// TIA Portal V18 export
// export: Created 2025-12-01T17:51:00.4461215Z, ExportSetting None, DisplayName Totally Integrated Automation Portal, DisplayVersion V18 Update 5, DisplayName TIA Portal Openness, DisplayVersion V18 Update 5, DisplayName TIA Portal Teamcenter Gateway, DisplayVersion V18, DisplayName TIA Portal Version Control Interface, DisplayVersion V18, DisplayName STEP 7 Professional, DisplayVersion V18 Update 5, DisplayName STEP 7 Safety, DisplayVersion V18, DisplayName WinCC Professional, DisplayVersion V18 Update 5
DATA_BLOCK "Parameter"   // DB170
{ S7_Optimized_Access := 'TRUE' }
// stored: AutoNumber false, IsRetainMemResEnabled true, MemoryReserve 10000
   VAR RETAIN
      AxisRun : Struct
         Axis : Array[1..15] of "ServoType_UDT";
      END_STRUCT;
      AxisNuw : Struct
         Axis : Array[1..15] of "ServoType_UDT";
      END_STRUCT;
      AxisDisplay : Struct
         Axis : Array[1..15] of "ServoType_UDT";
      END_STRUCT;
      AxisSave : Struct
         Axis : Array[1..15] of "ServoType_UDT";
      END_STRUCT;
      AxisStore : Array[1..15] of Struct
         Axis : Array[1..15] of "ServoType_UDT";
      END_STRUCT;
   END_VAR
BEGIN
   // AxisRun.Axis[1].Pos1 : 上料位1
   // AxisRun.Axis[2].Pos1 : 初始位
   // AxisRun.Axis[3].Pos1 : Home position / IV camera position 1
   // AxisRun.Axis[4].Pos1 : 上料位1
   // AxisRun.Axis[5].Pos1 : Z轴初始位
   // AxisRun.Axis[6].Pos1 : X轴初始位
   // AxisRun.Axis[7].Pos1 : Y轴初始位
   AxisRun.Axis[1].Pos1.Position := 3.12;
   AxisRun.Axis[2..3].Pos1.Position := 0.0;
   AxisRun.Axis[4].Pos1.Position := 3.585;
   AxisRun.Axis[5].Pos1.Position := 143.76;
   AxisRun.Axis[6].Pos1.Position := 2.34;
   AxisRun.Axis[7].Pos1.Position := 115.47;
   AxisRun.Axis[8..15].Pos1.Position := 0.0;
   AxisRun.Axis[1..2].Pos1.Speed := 10000;
   AxisRun.Axis[3].Pos1.Speed := 20000;
   AxisRun.Axis[4].Pos1.Speed := 10000;
   AxisRun.Axis[5..7].Pos1.Speed := 200;
   AxisRun.Axis[8..15].Pos1.Speed := 0;
   AxisRun.Axis[1..15].Pos1.Reached := FALSE;
   // AxisRun.Axis[1].Pos2 : 上料位2
   // AxisRun.Axis[2].Pos2 : 扫码位置2
   // AxisRun.Axis[3].Pos2 : Glue station 1 – end position
   // AxisRun.Axis[4].Pos2 : 上料位2
   // AxisRun.Axis[5].Pos2 : Z轴点胶位1
   // AxisRun.Axis[6].Pos2 : X轴点胶等待位
   // AxisRun.Axis[7].Pos2 : Y轴点胶位1
   AxisRun.Axis[1].Pos2.Position := 48.058;
   AxisRun.Axis[2].Pos2.Position := 45.0;
   AxisRun.Axis[3].Pos2.Position := 490.0;
   AxisRun.Axis[4].Pos2.Position := 48.61;
   AxisRun.Axis[5].Pos2.Position := 139.11;
   AxisRun.Axis[6].Pos2.Position := 76.0;
   AxisRun.Axis[7].Pos2.Position := 115.47;
   AxisRun.Axis[8..15].Pos2.Position := 0.0;
   AxisRun.Axis[1..2].Pos2.Speed := 10000;
   AxisRun.Axis[3].Pos2.Speed := 20000;
   AxisRun.Axis[4].Pos2.Speed := 10000;
   AxisRun.Axis[5..7].Pos2.Speed := 200;
   AxisRun.Axis[8..15].Pos2.Speed := 0;
   AxisRun.Axis[1..15].Pos2.Reached := FALSE;
   // AxisRun.Axis[1].Pos3 : 上料位3
   // AxisRun.Axis[2].Pos3 : 扫码位置3
   // AxisRun.Axis[3].Pos3 : Glue station 2 – end position
   // AxisRun.Axis[4].Pos3 : 上料位3
   // AxisRun.Axis[5].Pos3 : Z轴点胶位2
   // AxisRun.Axis[6].Pos3 : X轴点胶位1
   // AxisRun.Axis[7].Pos3 : Y轴点胶位2
   AxisRun.Axis[1].Pos3.Position := 93.154;
   AxisRun.Axis[2].Pos3.Position := 90.0;
   AxisRun.Axis[3].Pos3.Position := 490.0;
   AxisRun.Axis[4].Pos3.Position := 93.637;
   AxisRun.Axis[5].Pos3.Position := 131.98;
   AxisRun.Axis[6].Pos3.Position := 84.69;
   AxisRun.Axis[7].Pos3.Position := 115.47;
   AxisRun.Axis[8..15].Pos3.Position := 0.0;
   AxisRun.Axis[1..2].Pos3.Speed := 10000;
   AxisRun.Axis[3].Pos3.Speed := 20000;
   AxisRun.Axis[4].Pos3.Speed := 10000;
   AxisRun.Axis[5..7].Pos3.Speed := 200;
   AxisRun.Axis[8..15].Pos3.Speed := 0;
   AxisRun.Axis[1..15].Pos3.Reached := FALSE;
   // AxisRun.Axis[1].Pos4 : 上料位4
   // AxisRun.Axis[2].Pos4 : 扫码位置4
   // AxisRun.Axis[3].Pos4 : Glue station 3 – end position
   // AxisRun.Axis[4].Pos4 : 上料位4
   // AxisRun.Axis[5].Pos4 : Z轴点胶位3
   // AxisRun.Axis[6].Pos4 : X轴点胶位2
   // AxisRun.Axis[7].Pos4 : Y轴点胶位3
   AxisRun.Axis[1].Pos4.Position := 138.111;
   AxisRun.Axis[2].Pos4.Position := 135.0;
   AxisRun.Axis[3].Pos4.Position := 490.0;
   AxisRun.Axis[4].Pos4.Position := 138.606;
   AxisRun.Axis[5].Pos4.Position := 127.89;
   AxisRun.Axis[6].Pos4.Position := 84.69;
   AxisRun.Axis[7].Pos4.Position := 115.47;
   AxisRun.Axis[8..15].Pos4.Position := 0.0;
   AxisRun.Axis[1..2].Pos4.Speed := 10000;
   AxisRun.Axis[3].Pos4.Speed := 20000;
   AxisRun.Axis[4].Pos4.Speed := 10000;
   AxisRun.Axis[5..7].Pos4.Speed := 200;
   AxisRun.Axis[8..15].Pos4.Speed := 0;
   AxisRun.Axis[1..15].Pos4.Reached := FALSE;
   // AxisRun.Axis[1].Pos5 : 上料位5
   // AxisRun.Axis[2].Pos5 : 扫码位置5
   // AxisRun.Axis[3].Pos5 : Glue station 4 – end position // glue position cancelled
   // AxisRun.Axis[4].Pos5 : 上料位5
   // AxisRun.Axis[5].Pos5 : Z轴点胶位4
   // AxisRun.Axis[6].Pos5 : X轴点胶位3
   // AxisRun.Axis[7].Pos5 : Y轴点胶位4
   AxisRun.Axis[1].Pos5.Position := 183.025;
   AxisRun.Axis[2].Pos5.Position := 180.0;
   AxisRun.Axis[3].Pos5.Position := 0.0;
   AxisRun.Axis[4].Pos5.Position := 183.388;
   AxisRun.Axis[5].Pos5.Position := 0.0;
   AxisRun.Axis[6].Pos5.Position := 84.69;
   AxisRun.Axis[7].Pos5.Position := 115.47;
   AxisRun.Axis[8..15].Pos5.Position := 0.0;
   AxisRun.Axis[1..2].Pos5.Speed := 10000;
   AxisRun.Axis[3].Pos5.Speed := 0;
   AxisRun.Axis[4].Pos5.Speed := 10000;
   AxisRun.Axis[5].Pos5.Speed := 0;
   AxisRun.Axis[6..7].Pos5.Speed := 200;
   AxisRun.Axis[8..15].Pos5.Speed := 0;
   AxisRun.Axis[1..15].Pos5.Reached := FALSE;
   // AxisRun.Axis[1].Pos6 : 上料位6
   // AxisRun.Axis[2].Pos6 : 扫码位置6
   // AxisRun.Axis[3].Pos6 : Glue station 5 – end position
   // AxisRun.Axis[4].Pos6 : 上料位6
   // AxisRun.Axis[5].Pos6 : Z轴点胶位5
   // AxisRun.Axis[6].Pos6 : X轴点胶位4
   // AxisRun.Axis[7].Pos6 : Y轴点胶位5
   AxisRun.Axis[1].Pos6.Position := 228.065;
   AxisRun.Axis[2].Pos6.Position := 225.0;
   AxisRun.Axis[3].Pos6.Position := 490.0;
   AxisRun.Axis[4].Pos6.Position := 228.458;
   AxisRun.Axis[5].Pos6.Position := 127.0;
   AxisRun.Axis[6].Pos6.Position := 84.69;
   AxisRun.Axis[7].Pos6.Position := 110.18;
   AxisRun.Axis[8..15].Pos6.Position := 0.0;
   AxisRun.Axis[1..2].Pos6.Speed := 10000;
   AxisRun.Axis[3].Pos6.Speed := 5000;
   AxisRun.Axis[4].Pos6.Speed := 10000;
   AxisRun.Axis[5..7].Pos6.Speed := 200;
   AxisRun.Axis[8..15].Pos6.Speed := 0;
   AxisRun.Axis[1..15].Pos6.Reached := FALSE;
   // AxisRun.Axis[1].Pos7 : 上料位7
   // AxisRun.Axis[2].Pos7 : 扫码位置7
   // AxisRun.Axis[3].Pos7 : IV camera position 2
   // AxisRun.Axis[4].Pos7 : 上料位7
   // AxisRun.Axis[5].Pos7 : Z轴相机检测位
   // AxisRun.Axis[6].Pos7 : X轴点胶位5
   // AxisRun.Axis[7].Pos7 : Y轴相机检测位
   AxisRun.Axis[1].Pos7.Position := 273.195;
   AxisRun.Axis[2].Pos7.Position := 270.0;
   AxisRun.Axis[3].Pos7.Position := 90.0;
   AxisRun.Axis[4].Pos7.Position := 273.513;
   AxisRun.Axis[5].Pos7.Position := 48.11;
   AxisRun.Axis[6].Pos7.Position := 85.0;
   AxisRun.Axis[7].Pos7.Position := 60.52;
   AxisRun.Axis[8..15].Pos7.Position := 0.0;
   AxisRun.Axis[1..2].Pos7.Speed := 10000;
   AxisRun.Axis[3].Pos7.Speed := 20000;
   AxisRun.Axis[4].Pos7.Speed := 10000;
   AxisRun.Axis[5..7].Pos7.Speed := 200;
   AxisRun.Axis[8..15].Pos7.Speed := 0;
   AxisRun.Axis[1..15].Pos7.Reached := FALSE;
   // AxisRun.Axis[1].Pos8 : 上料位8
   // AxisRun.Axis[2].Pos8 : 扫码位置8
   // AxisRun.Axis[3].Pos8 : IV camera position 3
   // AxisRun.Axis[4].Pos8 : 上料位8
   // AxisRun.Axis[5].Pos8 : Z轴原点位
   // AxisRun.Axis[6].Pos8 : X轴相机检测位
   AxisRun.Axis[1].Pos8.Position := 318.05;
   AxisRun.Axis[2].Pos8.Position := 315.0;
   AxisRun.Axis[3].Pos8.Position := 180.0;
   AxisRun.Axis[4].Pos8.Position := 318.501;
   AxisRun.Axis[5].Pos8.Position := 0.0;
   AxisRun.Axis[6].Pos8.Position := 88.53;
   AxisRun.Axis[7].Pos8.Position := 80.0;
   AxisRun.Axis[8..15].Pos8.Position := 0.0;
   AxisRun.Axis[1..2].Pos8.Speed := 10000;
   AxisRun.Axis[3].Pos8.Speed := 20000;
   AxisRun.Axis[4].Pos8.Speed := 10000;
   AxisRun.Axis[5..6].Pos8.Speed := 200;
   AxisRun.Axis[7].Pos8.Speed := 100;
   AxisRun.Axis[8..15].Pos8.Speed := 0;
   AxisRun.Axis[1..15].Pos8.Reached := FALSE;
   // AxisRun.Axis[3].Pos9 : IV camera position 4
   // AxisRun.Axis[5].Pos9 : Z轴Up点胶位5
   AxisRun.Axis[1..2].Pos9.Position := 0.0;
   AxisRun.Axis[3].Pos9.Position := 270.0;
   AxisRun.Axis[4].Pos9.Position := 0.0;
   AxisRun.Axis[5].Pos9.Position := 48.11;
   AxisRun.Axis[6..15].Pos9.Position := 0.0;
   AxisRun.Axis[1..2].Pos9.Speed := 0;
   AxisRun.Axis[3].Pos9.Speed := 20000;
   AxisRun.Axis[4].Pos9.Speed := 0;
   AxisRun.Axis[5].Pos9.Speed := 200;
   AxisRun.Axis[6..15].Pos9.Speed := 0;
   AxisRun.Axis[1..15].Pos9.Reached := FALSE;
   AxisRun.Axis[1..15].Pos10.Position := 0.0;
   AxisRun.Axis[1..15].Pos10.Speed := 0;
   AxisRun.Axis[1..15].Pos10.Reached := FALSE;
   AxisRun.Axis[1..15].Pos11.Position := 0.0;
   AxisRun.Axis[1..15].Pos11.Speed := 0;
   AxisRun.Axis[1..15].Pos11.Reached := FALSE;
   AxisRun.Axis[1..15].Pos12.Position := 0.0;
   AxisRun.Axis[1..15].Pos12.Speed := 0;
   AxisRun.Axis[1..15].Pos12.Reached := FALSE;
   AxisRun.Axis[1..15].Pos13.Position := 0.0;
   AxisRun.Axis[1..15].Pos13.Speed := 0;
   AxisRun.Axis[1..15].Pos13.Reached := FALSE;
   AxisRun.Axis[1..15].Pos14.Position := 0.0;
   AxisRun.Axis[1..15].Pos14.Speed := 0;
   AxisRun.Axis[1..15].Pos14.Reached := FALSE;
   AxisRun.Axis[1..15].Pos15.Position := 0.0;
   AxisRun.Axis[1..15].Pos15.Speed := 0;
   AxisRun.Axis[1..15].Pos15.Reached := FALSE;
   AxisRun.Axis[1..15].Pos16.Position := 0.0;
   AxisRun.Axis[1..15].Pos16.Speed := 0;
   AxisRun.Axis[1..15].Pos16.Reached := FALSE;
   AxisRun.Axis[1..15].Pos17.Position := 0.0;
   AxisRun.Axis[1..15].Pos17.Speed := 0;
   AxisRun.Axis[1..15].Pos17.Reached := FALSE;
   AxisRun.Axis[1..15].Pos18.Position := 0.0;
   AxisRun.Axis[1..15].Pos18.Speed := 0;
   AxisRun.Axis[1..15].Pos18.Reached := FALSE;
   AxisRun.Axis[1..15].Pos19.Position := 0.0;
   AxisRun.Axis[1..15].Pos19.Speed := 0;
   AxisRun.Axis[1..15].Pos19.Reached := FALSE;
   AxisRun.Axis[1..15].Pos20.Position := 0.0;
   AxisRun.Axis[1..15].Pos20.Speed := 0;
   AxisRun.Axis[1..15].Pos20.Reached := FALSE;
   AxisRun.Axis[1..15].Pos21.Position := 0.0;
   AxisRun.Axis[1..15].Pos21.Speed := 0;
   AxisRun.Axis[1..15].Pos21.Reached := FALSE;
   AxisRun.Axis[1..15].Pos22.Position := 0.0;
   AxisRun.Axis[1..15].Pos22.Speed := 0;
   AxisRun.Axis[1..15].Pos22.Reached := FALSE;
   AxisRun.Axis[1..15].Pos23.Position := 0.0;
   AxisRun.Axis[1..15].Pos23.Speed := 0;
   AxisRun.Axis[1..15].Pos23.Reached := FALSE;
   AxisRun.Axis[1..15].Pos24.Position := 0.0;
   AxisRun.Axis[1..15].Pos24.Speed := 0;
   AxisRun.Axis[1..15].Pos24.Reached := FALSE;
   AxisRun.Axis[1..15].Pos25.Position := 0.0;
   AxisRun.Axis[1..15].Pos25.Speed := 0;
   AxisRun.Axis[1..15].Pos25.Reached := FALSE;
   AxisRun.Axis[1..15].Pos26.Position := 0.0;
   AxisRun.Axis[1..15].Pos26.Speed := 0;
   AxisRun.Axis[1..15].Pos26.Reached := FALSE;
   AxisRun.Axis[1..15].Pos27.Position := 0.0;
   AxisRun.Axis[1..15].Pos27.Speed := 0;
   AxisRun.Axis[1..15].Pos27.Reached := FALSE;
   AxisRun.Axis[1..15].Pos28.Position := 0.0;
   AxisRun.Axis[1..15].Pos28.Speed := 0;
   AxisRun.Axis[1..15].Pos28.Reached := FALSE;
   AxisRun.Axis[1..15].Pos29.Position := 0.0;
   AxisRun.Axis[1..15].Pos29.Speed := 0;
   AxisRun.Axis[1..15].Pos29.Reached := FALSE;
   AxisRun.Axis[1..15].Pos30.Position := 0.0;
   AxisRun.Axis[1..15].Pos30.Speed := 0;
   AxisRun.Axis[1..15].Pos30.Reached := FALSE;
   AxisNuw.Axis[1..15].Pos1.Position := 0.0;
   AxisNuw.Axis[1..15].Pos1.Speed := 0;
   AxisNuw.Axis[1..15].Pos1.Reached := FALSE;
   AxisNuw.Axis[1..15].Pos2.Position := 0.0;
   AxisNuw.Axis[1..15].Pos2.Speed := 0;
   AxisNuw.Axis[1..15].Pos2.Reached := FALSE;
   AxisNuw.Axis[1..15].Pos3.Position := 0.0;
   AxisNuw.Axis[1..15].Pos3.Speed := 0;
   AxisNuw.Axis[1..15].Pos3.Reached := FALSE;
   AxisNuw.Axis[1..15].Pos4.Position := 0.0;
   AxisNuw.Axis[1..15].Pos4.Speed := 0;
   AxisNuw.Axis[1..15].Pos4.Reached := FALSE;
   AxisNuw.Axis[1..15].Pos5.Position := 0.0;
   AxisNuw.Axis[1..15].Pos5.Speed := 0;
   AxisNuw.Axis[1..15].Pos5.Reached := FALSE;
   AxisNuw.Axis[1..15].Pos6.Position := 0.0;
   AxisNuw.Axis[1..15].Pos6.Speed := 0;
   AxisNuw.Axis[1..15].Pos6.Reached := FALSE;
   AxisNuw.Axis[1..15].Pos7.Position := 0.0;
   AxisNuw.Axis[1..15].Pos7.Speed := 0;
   AxisNuw.Axis[1..15].Pos7.Reached := FALSE;
   AxisNuw.Axis[1..15].Pos8.Position := 0.0;
   AxisNuw.Axis[1..15].Pos8.Speed := 0;
   AxisNuw.Axis[1..15].Pos8.Reached := FALSE;
   AxisNuw.Axis[1..15].Pos9.Position := 0.0;
   AxisNuw.Axis[1..15].Pos9.Speed := 0;
   AxisNuw.Axis[1..15].Pos9.Reached := FALSE;
   AxisNuw.Axis[1..15].Pos10.Position := 0.0;
   AxisNuw.Axis[1..15].Pos10.Speed := 0;
   AxisNuw.Axis[1..15].Pos10.Reached := FALSE;
   AxisNuw.Axis[1..15].Pos11.Position := 0.0;
   AxisNuw.Axis[1..15].Pos11.Speed := 0;
   AxisNuw.Axis[1..15].Pos11.Reached := FALSE;
   AxisNuw.Axis[1..15].Pos12.Position := 0.0;
   AxisNuw.Axis[1..15].Pos12.Speed := 0;
   AxisNuw.Axis[1..15].Pos12.Reached := FALSE;
   AxisNuw.Axis[1..15].Pos13.Position := 0.0;
   AxisNuw.Axis[1..15].Pos13.Speed := 0;
   AxisNuw.Axis[1..15].Pos13.Reached := FALSE;
   AxisNuw.Axis[1..15].Pos14.Position := 0.0;
   AxisNuw.Axis[1..15].Pos14.Speed := 0;
   AxisNuw.Axis[1..15].Pos14.Reached := FALSE;
   AxisNuw.Axis[1..15].Pos15.Position := 0.0;
   AxisNuw.Axis[1..15].Pos15.Speed := 0;
   AxisNuw.Axis[1..15].Pos15.Reached := FALSE;
   AxisNuw.Axis[1..15].Pos16.Position := 0.0;
   AxisNuw.Axis[1..15].Pos16.Speed := 0;
   AxisNuw.Axis[1..15].Pos16.Reached := FALSE;
   AxisNuw.Axis[1..15].Pos17.Position := 0.0;
   AxisNuw.Axis[1..15].Pos17.Speed := 0;
   AxisNuw.Axis[1..15].Pos17.Reached := FALSE;
   AxisNuw.Axis[1..15].Pos18.Position := 0.0;
   AxisNuw.Axis[1..15].Pos18.Speed := 0;
   AxisNuw.Axis[1..15].Pos18.Reached := FALSE;
   AxisNuw.Axis[1..15].Pos19.Position := 0.0;
   AxisNuw.Axis[1..15].Pos19.Speed := 0;
   AxisNuw.Axis[1..15].Pos19.Reached := FALSE;
   AxisNuw.Axis[1..15].Pos20.Position := 0.0;
   AxisNuw.Axis[1..15].Pos20.Speed := 0;
   AxisNuw.Axis[1..15].Pos20.Reached := FALSE;
   AxisNuw.Axis[1..15].Pos21.Position := 0.0;
   AxisNuw.Axis[1..15].Pos21.Speed := 0;
   AxisNuw.Axis[1..15].Pos21.Reached := FALSE;
   AxisNuw.Axis[1..15].Pos22.Position := 0.0;
   AxisNuw.Axis[1..15].Pos22.Speed := 0;
   AxisNuw.Axis[1..15].Pos22.Reached := FALSE;
   AxisNuw.Axis[1..15].Pos23.Position := 0.0;
   AxisNuw.Axis[1..15].Pos23.Speed := 0;
   AxisNuw.Axis[1..15].Pos23.Reached := FALSE;
   AxisNuw.Axis[1..15].Pos24.Position := 0.0;
   AxisNuw.Axis[1..15].Pos24.Speed := 0;
   AxisNuw.Axis[1..15].Pos24.Reached := FALSE;
   AxisNuw.Axis[1..15].Pos25.Position := 0.0;
   AxisNuw.Axis[1..15].Pos25.Speed := 0;
   AxisNuw.Axis[1..15].Pos25.Reached := FALSE;
   AxisNuw.Axis[1..15].Pos26.Position := 0.0;
   AxisNuw.Axis[1..15].Pos26.Speed := 0;
   AxisNuw.Axis[1..15].Pos26.Reached := FALSE;
   AxisNuw.Axis[1..15].Pos27.Position := 0.0;
   AxisNuw.Axis[1..15].Pos27.Speed := 0;
   AxisNuw.Axis[1..15].Pos27.Reached := FALSE;
   AxisNuw.Axis[1..15].Pos28.Position := 0.0;
   AxisNuw.Axis[1..15].Pos28.Speed := 0;
   AxisNuw.Axis[1..15].Pos28.Reached := FALSE;
   AxisNuw.Axis[1..15].Pos29.Position := 0.0;
   AxisNuw.Axis[1..15].Pos29.Speed := 0;
   AxisNuw.Axis[1..15].Pos29.Reached := FALSE;
   AxisNuw.Axis[1..15].Pos30.Position := 0.0;
   AxisNuw.Axis[1..15].Pos30.Speed := 0;
   AxisNuw.Axis[1..15].Pos30.Reached := FALSE;
   AxisDisplay.Axis[1..15].Pos1.Position := 0.0;
   AxisDisplay.Axis[1..15].Pos1.Speed := 0;
   AxisDisplay.Axis[1..15].Pos1.Reached := FALSE;
   AxisDisplay.Axis[1..15].Pos2.Position := 0.0;
   AxisDisplay.Axis[1..15].Pos2.Speed := 0;
   AxisDisplay.Axis[1..15].Pos2.Reached := FALSE;
   AxisDisplay.Axis[1..15].Pos3.Position := 0.0;
   AxisDisplay.Axis[1..15].Pos3.Speed := 0;
   AxisDisplay.Axis[1..15].Pos3.Reached := FALSE;
   AxisDisplay.Axis[1..15].Pos4.Position := 0.0;
   AxisDisplay.Axis[1..15].Pos4.Speed := 0;
   AxisDisplay.Axis[1..15].Pos4.Reached := FALSE;
   AxisDisplay.Axis[1..15].Pos5.Position := 0.0;
   AxisDisplay.Axis[1..15].Pos5.Speed := 0;
   AxisDisplay.Axis[1..15].Pos5.Reached := FALSE;
   AxisDisplay.Axis[1..15].Pos6.Position := 0.0;
   AxisDisplay.Axis[1..15].Pos6.Speed := 0;
   AxisDisplay.Axis[1..15].Pos6.Reached := FALSE;
   AxisDisplay.Axis[1..15].Pos7.Position := 0.0;
   AxisDisplay.Axis[1..15].Pos7.Speed := 0;
   AxisDisplay.Axis[1..15].Pos7.Reached := FALSE;
   AxisDisplay.Axis[1..15].Pos8.Position := 0.0;
   AxisDisplay.Axis[1..15].Pos8.Speed := 0;
   AxisDisplay.Axis[1..15].Pos8.Reached := FALSE;
   AxisDisplay.Axis[1..15].Pos9.Position := 0.0;
   AxisDisplay.Axis[1..15].Pos9.Speed := 0;
   AxisDisplay.Axis[1..15].Pos9.Reached := FALSE;
   AxisDisplay.Axis[1..15].Pos10.Position := 0.0;
   AxisDisplay.Axis[1..15].Pos10.Speed := 0;
   AxisDisplay.Axis[1..15].Pos10.Reached := FALSE;
   AxisDisplay.Axis[1..15].Pos11.Position := 0.0;
   AxisDisplay.Axis[1..15].Pos11.Speed := 0;
   AxisDisplay.Axis[1..15].Pos11.Reached := FALSE;
   AxisDisplay.Axis[1..15].Pos12.Position := 0.0;
   AxisDisplay.Axis[1..15].Pos12.Speed := 0;
   AxisDisplay.Axis[1..15].Pos12.Reached := FALSE;
   AxisDisplay.Axis[1..15].Pos13.Position := 0.0;
   AxisDisplay.Axis[1..15].Pos13.Speed := 0;
   AxisDisplay.Axis[1..15].Pos13.Reached := FALSE;
   AxisDisplay.Axis[1..15].Pos14.Position := 0.0;
   AxisDisplay.Axis[1..15].Pos14.Speed := 0;
   AxisDisplay.Axis[1..15].Pos14.Reached := FALSE;
   AxisDisplay.Axis[1..15].Pos15.Position := 0.0;
   AxisDisplay.Axis[1..15].Pos15.Speed := 0;
   AxisDisplay.Axis[1..15].Pos15.Reached := FALSE;
   AxisDisplay.Axis[1..15].Pos16.Position := 0.0;
   AxisDisplay.Axis[1..15].Pos16.Speed := 0;
   AxisDisplay.Axis[1..15].Pos16.Reached := FALSE;
   AxisDisplay.Axis[1..15].Pos17.Position := 0.0;
   AxisDisplay.Axis[1..15].Pos17.Speed := 0;
   AxisDisplay.Axis[1..15].Pos17.Reached := FALSE;
   AxisDisplay.Axis[1..15].Pos18.Position := 0.0;
   AxisDisplay.Axis[1..15].Pos18.Speed := 0;
   AxisDisplay.Axis[1..15].Pos18.Reached := FALSE;
   AxisDisplay.Axis[1..15].Pos19.Position := 0.0;
   AxisDisplay.Axis[1..15].Pos19.Speed := 0;
   AxisDisplay.Axis[1..15].Pos19.Reached := FALSE;
   AxisDisplay.Axis[1..15].Pos20.Position := 0.0;
   AxisDisplay.Axis[1..15].Pos20.Speed := 0;
   AxisDisplay.Axis[1..15].Pos20.Reached := FALSE;
   AxisDisplay.Axis[1..15].Pos21.Position := 0.0;
   AxisDisplay.Axis[1..15].Pos21.Speed := 0;
   AxisDisplay.Axis[1..15].Pos21.Reached := FALSE;
   AxisDisplay.Axis[1..15].Pos22.Position := 0.0;
   AxisDisplay.Axis[1..15].Pos22.Speed := 0;
   AxisDisplay.Axis[1..15].Pos22.Reached := FALSE;
   AxisDisplay.Axis[1..15].Pos23.Position := 0.0;
   AxisDisplay.Axis[1..15].Pos23.Speed := 0;
   AxisDisplay.Axis[1..15].Pos23.Reached := FALSE;
   AxisDisplay.Axis[1..15].Pos24.Position := 0.0;
   AxisDisplay.Axis[1..15].Pos24.Speed := 0;
   AxisDisplay.Axis[1..15].Pos24.Reached := FALSE;
   AxisDisplay.Axis[1..15].Pos25.Position := 0.0;
   AxisDisplay.Axis[1..15].Pos25.Speed := 0;
   AxisDisplay.Axis[1..15].Pos25.Reached := FALSE;
   AxisDisplay.Axis[1..15].Pos26.Position := 0.0;
   AxisDisplay.Axis[1..15].Pos26.Speed := 0;
   AxisDisplay.Axis[1..15].Pos26.Reached := FALSE;
   AxisDisplay.Axis[1..15].Pos27.Position := 0.0;
   AxisDisplay.Axis[1..15].Pos27.Speed := 0;
   AxisDisplay.Axis[1..15].Pos27.Reached := FALSE;
   AxisDisplay.Axis[1..15].Pos28.Position := 0.0;
   AxisDisplay.Axis[1..15].Pos28.Speed := 0;
   AxisDisplay.Axis[1..15].Pos28.Reached := FALSE;
   AxisDisplay.Axis[1..15].Pos29.Position := 0.0;
   AxisDisplay.Axis[1..15].Pos29.Speed := 0;
   AxisDisplay.Axis[1..15].Pos29.Reached := FALSE;
   AxisDisplay.Axis[1..15].Pos30.Position := 0.0;
   AxisDisplay.Axis[1..15].Pos30.Speed := 0;
   AxisDisplay.Axis[1..15].Pos30.Reached := FALSE;
   AxisSave.Axis[1..15].Pos1.Position := 0.0;
   AxisSave.Axis[1..15].Pos1.Speed := 0;
   AxisSave.Axis[1..15].Pos1.Reached := FALSE;
   AxisSave.Axis[1..15].Pos2.Position := 0.0;
   AxisSave.Axis[1..15].Pos2.Speed := 0;
   AxisSave.Axis[1..15].Pos2.Reached := FALSE;
   AxisSave.Axis[1..15].Pos3.Position := 0.0;
   AxisSave.Axis[1..15].Pos3.Speed := 0;
   AxisSave.Axis[1..15].Pos3.Reached := FALSE;
   AxisSave.Axis[1..15].Pos4.Position := 0.0;
   AxisSave.Axis[1..15].Pos4.Speed := 0;
   AxisSave.Axis[1..15].Pos4.Reached := FALSE;
   AxisSave.Axis[1..15].Pos5.Position := 0.0;
   AxisSave.Axis[1..15].Pos5.Speed := 0;
   AxisSave.Axis[1..15].Pos5.Reached := FALSE;
   AxisSave.Axis[1..15].Pos6.Position := 0.0;
   AxisSave.Axis[1..15].Pos6.Speed := 0;
   AxisSave.Axis[1..15].Pos6.Reached := FALSE;
   AxisSave.Axis[1..15].Pos7.Position := 0.0;
   AxisSave.Axis[1..15].Pos7.Speed := 0;
   AxisSave.Axis[1..15].Pos7.Reached := FALSE;
   AxisSave.Axis[1..15].Pos8.Position := 0.0;
   AxisSave.Axis[1..15].Pos8.Speed := 0;
   AxisSave.Axis[1..15].Pos8.Reached := FALSE;
   AxisSave.Axis[1..15].Pos9.Position := 0.0;
   AxisSave.Axis[1..15].Pos9.Speed := 0;
   AxisSave.Axis[1..15].Pos9.Reached := FALSE;
   AxisSave.Axis[1..15].Pos10.Position := 0.0;
   AxisSave.Axis[1..15].Pos10.Speed := 0;
   AxisSave.Axis[1..15].Pos10.Reached := FALSE;
   AxisSave.Axis[1..15].Pos11.Position := 0.0;
   AxisSave.Axis[1..15].Pos11.Speed := 0;
   AxisSave.Axis[1..15].Pos11.Reached := FALSE;
   AxisSave.Axis[1..15].Pos12.Position := 0.0;
   AxisSave.Axis[1..15].Pos12.Speed := 0;
   AxisSave.Axis[1..15].Pos12.Reached := FALSE;
   AxisSave.Axis[1..15].Pos13.Position := 0.0;
   AxisSave.Axis[1..15].Pos13.Speed := 0;
   AxisSave.Axis[1..15].Pos13.Reached := FALSE;
   AxisSave.Axis[1..15].Pos14.Position := 0.0;
   AxisSave.Axis[1..15].Pos14.Speed := 0;
   AxisSave.Axis[1..15].Pos14.Reached := FALSE;
   AxisSave.Axis[1..15].Pos15.Position := 0.0;
   AxisSave.Axis[1..15].Pos15.Speed := 0;
   AxisSave.Axis[1..15].Pos15.Reached := FALSE;
   AxisSave.Axis[1..15].Pos16.Position := 0.0;
   AxisSave.Axis[1..15].Pos16.Speed := 0;
   AxisSave.Axis[1..15].Pos16.Reached := FALSE;
   AxisSave.Axis[1..15].Pos17.Position := 0.0;
   AxisSave.Axis[1..15].Pos17.Speed := 0;
   AxisSave.Axis[1..15].Pos17.Reached := FALSE;
   AxisSave.Axis[1..15].Pos18.Position := 0.0;
   AxisSave.Axis[1..15].Pos18.Speed := 0;
   AxisSave.Axis[1..15].Pos18.Reached := FALSE;
   AxisSave.Axis[1..15].Pos19.Position := 0.0;
   AxisSave.Axis[1..15].Pos19.Speed := 0;
   AxisSave.Axis[1..15].Pos19.Reached := FALSE;
   AxisSave.Axis[1..15].Pos20.Position := 0.0;
   AxisSave.Axis[1..15].Pos20.Speed := 0;
   AxisSave.Axis[1..15].Pos20.Reached := FALSE;
   AxisSave.Axis[1..15].Pos21.Position := 0.0;
   AxisSave.Axis[1..15].Pos21.Speed := 0;
   AxisSave.Axis[1..15].Pos21.Reached := FALSE;
   AxisSave.Axis[1..15].Pos22.Position := 0.0;
   AxisSave.Axis[1..15].Pos22.Speed := 0;
   AxisSave.Axis[1..15].Pos22.Reached := FALSE;
   AxisSave.Axis[1..15].Pos23.Position := 0.0;
   AxisSave.Axis[1..15].Pos23.Speed := 0;
   AxisSave.Axis[1..15].Pos23.Reached := FALSE;
   AxisSave.Axis[1..15].Pos24.Position := 0.0;
   AxisSave.Axis[1..15].Pos24.Speed := 0;
   AxisSave.Axis[1..15].Pos24.Reached := FALSE;
   AxisSave.Axis[1..15].Pos25.Position := 0.0;
   AxisSave.Axis[1..15].Pos25.Speed := 0;
   AxisSave.Axis[1..15].Pos25.Reached := FALSE;
   AxisSave.Axis[1..15].Pos26.Position := 0.0;
   AxisSave.Axis[1..15].Pos26.Speed := 0;
   AxisSave.Axis[1..15].Pos26.Reached := FALSE;
   AxisSave.Axis[1..15].Pos27.Position := 0.0;
   AxisSave.Axis[1..15].Pos27.Speed := 0;
   AxisSave.Axis[1..15].Pos27.Reached := FALSE;
   AxisSave.Axis[1..15].Pos28.Position := 0.0;
   AxisSave.Axis[1..15].Pos28.Speed := 0;
   AxisSave.Axis[1..15].Pos28.Reached := FALSE;
   AxisSave.Axis[1..15].Pos29.Position := 0.0;
   AxisSave.Axis[1..15].Pos29.Speed := 0;
   AxisSave.Axis[1..15].Pos29.Reached := FALSE;
   AxisSave.Axis[1..15].Pos30.Position := 0.0;
   AxisSave.Axis[1..15].Pos30.Speed := 0;
   AxisSave.Axis[1..15].Pos30.Reached := FALSE;
   AxisStore[1].Axis[1..15].Pos1.Position := 0.0;
   AxisStore[2].Axis[1..15].Pos1.Position := 0.0;
   AxisStore[3].Axis[1..15].Pos1.Position := 0.0;
   AxisStore[4].Axis[1..15].Pos1.Position := 0.0;
   AxisStore[5].Axis[1..15].Pos1.Position := 0.0;
   AxisStore[6].Axis[1..15].Pos1.Position := 0.0;
   AxisStore[7].Axis[1..15].Pos1.Position := 0.0;
   AxisStore[8].Axis[1..15].Pos1.Position := 0.0;
   AxisStore[9].Axis[1..15].Pos1.Position := 0.0;
   AxisStore[10].Axis[1..15].Pos1.Position := 0.0;
   AxisStore[11].Axis[1..15].Pos1.Position := 0.0;
   AxisStore[12].Axis[1..15].Pos1.Position := 0.0;
   AxisStore[13].Axis[1..15].Pos1.Position := 0.0;
   AxisStore[14].Axis[1..15].Pos1.Position := 0.0;
   AxisStore[15].Axis[1..15].Pos1.Position := 0.0;
   AxisStore[1].Axis[1..15].Pos1.Speed := 0;
   AxisStore[2].Axis[1..15].Pos1.Speed := 0;
   AxisStore[3].Axis[1..15].Pos1.Speed := 0;
   AxisStore[4].Axis[1..15].Pos1.Speed := 0;
   AxisStore[5].Axis[1..15].Pos1.Speed := 0;
   AxisStore[6].Axis[1..15].Pos1.Speed := 0;
   AxisStore[7].Axis[1..15].Pos1.Speed := 0;
   AxisStore[8].Axis[1..15].Pos1.Speed := 0;
   AxisStore[9].Axis[1..15].Pos1.Speed := 0;
   AxisStore[10].Axis[1..15].Pos1.Speed := 0;
   AxisStore[11].Axis[1..15].Pos1.Speed := 0;
   AxisStore[12].Axis[1..15].Pos1.Speed := 0;
   AxisStore[13].Axis[1..15].Pos1.Speed := 0;
   AxisStore[14].Axis[1..15].Pos1.Speed := 0;
   AxisStore[15].Axis[1..15].Pos1.Speed := 0;
   AxisStore[1].Axis[1..15].Pos1.Reached := FALSE;
   AxisStore[2].Axis[1..15].Pos1.Reached := FALSE;
   AxisStore[3].Axis[1..15].Pos1.Reached := FALSE;
   AxisStore[4].Axis[1..15].Pos1.Reached := FALSE;
   AxisStore[5].Axis[1..15].Pos1.Reached := FALSE;
   AxisStore[6].Axis[1..15].Pos1.Reached := FALSE;
   AxisStore[7].Axis[1..15].Pos1.Reached := FALSE;
   AxisStore[8].Axis[1..15].Pos1.Reached := FALSE;
   AxisStore[9].Axis[1..15].Pos1.Reached := FALSE;
   AxisStore[10].Axis[1..15].Pos1.Reached := FALSE;
   AxisStore[11].Axis[1..15].Pos1.Reached := FALSE;
   AxisStore[12].Axis[1..15].Pos1.Reached := FALSE;
   AxisStore[13].Axis[1..15].Pos1.Reached := FALSE;
   AxisStore[14].Axis[1..15].Pos1.Reached := FALSE;
   AxisStore[15].Axis[1..15].Pos1.Reached := FALSE;
   AxisStore[1].Axis[1..15].Pos2.Position := 0.0;
   AxisStore[2].Axis[1..15].Pos2.Position := 0.0;
   AxisStore[3].Axis[1..15].Pos2.Position := 0.0;
   AxisStore[4].Axis[1..15].Pos2.Position := 0.0;
   AxisStore[5].Axis[1..15].Pos2.Position := 0.0;
   AxisStore[6].Axis[1..15].Pos2.Position := 0.0;
   AxisStore[7].Axis[1..15].Pos2.Position := 0.0;
   AxisStore[8].Axis[1..15].Pos2.Position := 0.0;
   AxisStore[9].Axis[1..15].Pos2.Position := 0.0;
   AxisStore[10].Axis[1..15].Pos2.Position := 0.0;
   AxisStore[11].Axis[1..15].Pos2.Position := 0.0;
   AxisStore[12].Axis[1..15].Pos2.Position := 0.0;
   AxisStore[13].Axis[1..15].Pos2.Position := 0.0;
   AxisStore[14].Axis[1..15].Pos2.Position := 0.0;
   AxisStore[15].Axis[1..15].Pos2.Position := 0.0;
   AxisStore[1].Axis[1..15].Pos2.Speed := 0;
   AxisStore[2].Axis[1..15].Pos2.Speed := 0;
   AxisStore[3].Axis[1..15].Pos2.Speed := 0;
   AxisStore[4].Axis[1..15].Pos2.Speed := 0;
   AxisStore[5].Axis[1..15].Pos2.Speed := 0;
   AxisStore[6].Axis[1..15].Pos2.Speed := 0;
   AxisStore[7].Axis[1..15].Pos2.Speed := 0;
   AxisStore[8].Axis[1..15].Pos2.Speed := 0;
   AxisStore[9].Axis[1..15].Pos2.Speed := 0;
   AxisStore[10].Axis[1..15].Pos2.Speed := 0;
   AxisStore[11].Axis[1..15].Pos2.Speed := 0;
   AxisStore[12].Axis[1..15].Pos2.Speed := 0;
   AxisStore[13].Axis[1..15].Pos2.Speed := 0;
   AxisStore[14].Axis[1..15].Pos2.Speed := 0;
   AxisStore[15].Axis[1..15].Pos2.Speed := 0;
   AxisStore[1].Axis[1..15].Pos2.Reached := FALSE;
   AxisStore[2].Axis[1..15].Pos2.Reached := FALSE;
   AxisStore[3].Axis[1..15].Pos2.Reached := FALSE;
   AxisStore[4].Axis[1..15].Pos2.Reached := FALSE;
   AxisStore[5].Axis[1..15].Pos2.Reached := FALSE;
   AxisStore[6].Axis[1..15].Pos2.Reached := FALSE;
   AxisStore[7].Axis[1..15].Pos2.Reached := FALSE;
   AxisStore[8].Axis[1..15].Pos2.Reached := FALSE;
   AxisStore[9].Axis[1..15].Pos2.Reached := FALSE;
   AxisStore[10].Axis[1..15].Pos2.Reached := FALSE;
   AxisStore[11].Axis[1..15].Pos2.Reached := FALSE;
   AxisStore[12].Axis[1..15].Pos2.Reached := FALSE;
   AxisStore[13].Axis[1..15].Pos2.Reached := FALSE;
   AxisStore[14].Axis[1..15].Pos2.Reached := FALSE;
   AxisStore[15].Axis[1..15].Pos2.Reached := FALSE;
   AxisStore[1].Axis[1..15].Pos3.Position := 0.0;
   AxisStore[2].Axis[1..15].Pos3.Position := 0.0;
   AxisStore[3].Axis[1..15].Pos3.Position := 0.0;
   AxisStore[4].Axis[1..15].Pos3.Position := 0.0;
   AxisStore[5].Axis[1..15].Pos3.Position := 0.0;
   AxisStore[6].Axis[1..15].Pos3.Position := 0.0;
   AxisStore[7].Axis[1..15].Pos3.Position := 0.0;
   AxisStore[8].Axis[1..15].Pos3.Position := 0.0;
   AxisStore[9].Axis[1..15].Pos3.Position := 0.0;
   AxisStore[10].Axis[1..15].Pos3.Position := 0.0;
   AxisStore[11].Axis[1..15].Pos3.Position := 0.0;
   AxisStore[12].Axis[1..15].Pos3.Position := 0.0;
   AxisStore[13].Axis[1..15].Pos3.Position := 0.0;
   AxisStore[14].Axis[1..15].Pos3.Position := 0.0;
   AxisStore[15].Axis[1..15].Pos3.Position := 0.0;
   AxisStore[1].Axis[1..15].Pos3.Speed := 0;
   AxisStore[2].Axis[1..15].Pos3.Speed := 0;
   AxisStore[3].Axis[1..15].Pos3.Speed := 0;
   AxisStore[4].Axis[1..15].Pos3.Speed := 0;
   AxisStore[5].Axis[1..15].Pos3.Speed := 0;
   AxisStore[6].Axis[1..15].Pos3.Speed := 0;
   AxisStore[7].Axis[1..15].Pos3.Speed := 0;
   AxisStore[8].Axis[1..15].Pos3.Speed := 0;
   AxisStore[9].Axis[1..15].Pos3.Speed := 0;
   AxisStore[10].Axis[1..15].Pos3.Speed := 0;
   AxisStore[11].Axis[1..15].Pos3.Speed := 0;
   AxisStore[12].Axis[1..15].Pos3.Speed := 0;
   AxisStore[13].Axis[1..15].Pos3.Speed := 0;
   AxisStore[14].Axis[1..15].Pos3.Speed := 0;
   AxisStore[15].Axis[1..15].Pos3.Speed := 0;
   AxisStore[1].Axis[1..15].Pos3.Reached := FALSE;
   AxisStore[2].Axis[1..15].Pos3.Reached := FALSE;
   AxisStore[3].Axis[1..15].Pos3.Reached := FALSE;
   AxisStore[4].Axis[1..15].Pos3.Reached := FALSE;
   AxisStore[5].Axis[1..15].Pos3.Reached := FALSE;
   AxisStore[6].Axis[1..15].Pos3.Reached := FALSE;
   AxisStore[7].Axis[1..15].Pos3.Reached := FALSE;
   AxisStore[8].Axis[1..15].Pos3.Reached := FALSE;
   AxisStore[9].Axis[1..15].Pos3.Reached := FALSE;
   AxisStore[10].Axis[1..15].Pos3.Reached := FALSE;
   AxisStore[11].Axis[1..15].Pos3.Reached := FALSE;
   AxisStore[12].Axis[1..15].Pos3.Reached := FALSE;
   AxisStore[13].Axis[1..15].Pos3.Reached := FALSE;
   AxisStore[14].Axis[1..15].Pos3.Reached := FALSE;
   AxisStore[15].Axis[1..15].Pos3.Reached := FALSE;
   AxisStore[1].Axis[1..15].Pos4.Position := 0.0;
   AxisStore[2].Axis[1..15].Pos4.Position := 0.0;
   AxisStore[3].Axis[1..15].Pos4.Position := 0.0;
   AxisStore[4].Axis[1..15].Pos4.Position := 0.0;
   AxisStore[5].Axis[1..15].Pos4.Position := 0.0;
   AxisStore[6].Axis[1..15].Pos4.Position := 0.0;
   AxisStore[7].Axis[1..15].Pos4.Position := 0.0;
   AxisStore[8].Axis[1..15].Pos4.Position := 0.0;
   AxisStore[9].Axis[1..15].Pos4.Position := 0.0;
   AxisStore[10].Axis[1..15].Pos4.Position := 0.0;
   AxisStore[11].Axis[1..15].Pos4.Position := 0.0;
   AxisStore[12].Axis[1..15].Pos4.Position := 0.0;
   AxisStore[13].Axis[1..15].Pos4.Position := 0.0;
   AxisStore[14].Axis[1..15].Pos4.Position := 0.0;
   AxisStore[15].Axis[1..15].Pos4.Position := 0.0;
   AxisStore[1].Axis[1..15].Pos4.Speed := 0;
   AxisStore[2].Axis[1..15].Pos4.Speed := 0;
   AxisStore[3].Axis[1..15].Pos4.Speed := 0;
   AxisStore[4].Axis[1..15].Pos4.Speed := 0;
   AxisStore[5].Axis[1..15].Pos4.Speed := 0;
   AxisStore[6].Axis[1..15].Pos4.Speed := 0;
   AxisStore[7].Axis[1..15].Pos4.Speed := 0;
   AxisStore[8].Axis[1..15].Pos4.Speed := 0;
   AxisStore[9].Axis[1..15].Pos4.Speed := 0;
   AxisStore[10].Axis[1..15].Pos4.Speed := 0;
   AxisStore[11].Axis[1..15].Pos4.Speed := 0;
   AxisStore[12].Axis[1..15].Pos4.Speed := 0;
   AxisStore[13].Axis[1..15].Pos4.Speed := 0;
   AxisStore[14].Axis[1..15].Pos4.Speed := 0;
   AxisStore[15].Axis[1..15].Pos4.Speed := 0;
   AxisStore[1].Axis[1..15].Pos4.Reached := FALSE;
   AxisStore[2].Axis[1..15].Pos4.Reached := FALSE;
   AxisStore[3].Axis[1..15].Pos4.Reached := FALSE;
   AxisStore[4].Axis[1..15].Pos4.Reached := FALSE;
   AxisStore[5].Axis[1..15].Pos4.Reached := FALSE;
   AxisStore[6].Axis[1..15].Pos4.Reached := FALSE;
   AxisStore[7].Axis[1..15].Pos4.Reached := FALSE;
   AxisStore[8].Axis[1..15].Pos4.Reached := FALSE;
   AxisStore[9].Axis[1..15].Pos4.Reached := FALSE;
   AxisStore[10].Axis[1..15].Pos4.Reached := FALSE;
   AxisStore[11].Axis[1..15].Pos4.Reached := FALSE;
   AxisStore[12].Axis[1..15].Pos4.Reached := FALSE;
   AxisStore[13].Axis[1..15].Pos4.Reached := FALSE;
   AxisStore[14].Axis[1..15].Pos4.Reached := FALSE;
   AxisStore[15].Axis[1..15].Pos4.Reached := FALSE;
   AxisStore[1].Axis[1..15].Pos5.Position := 0.0;
   AxisStore[2].Axis[1..15].Pos5.Position := 0.0;
   AxisStore[3].Axis[1..15].Pos5.Position := 0.0;
   AxisStore[4].Axis[1..15].Pos5.Position := 0.0;
   AxisStore[5].Axis[1..15].Pos5.Position := 0.0;
   AxisStore[6].Axis[1..15].Pos5.Position := 0.0;
   AxisStore[7].Axis[1..15].Pos5.Position := 0.0;
   AxisStore[8].Axis[1..15].Pos5.Position := 0.0;
   AxisStore[9].Axis[1..15].Pos5.Position := 0.0;
   AxisStore[10].Axis[1..15].Pos5.Position := 0.0;
   AxisStore[11].Axis[1..15].Pos5.Position := 0.0;
   AxisStore[12].Axis[1..15].Pos5.Position := 0.0;
   AxisStore[13].Axis[1..15].Pos5.Position := 0.0;
   AxisStore[14].Axis[1..15].Pos5.Position := 0.0;
   AxisStore[15].Axis[1..15].Pos5.Position := 0.0;
   AxisStore[1].Axis[1..15].Pos5.Speed := 0;
   AxisStore[2].Axis[1..15].Pos5.Speed := 0;
   AxisStore[3].Axis[1..15].Pos5.Speed := 0;
   AxisStore[4].Axis[1..15].Pos5.Speed := 0;
   AxisStore[5].Axis[1..15].Pos5.Speed := 0;
   AxisStore[6].Axis[1..15].Pos5.Speed := 0;
   AxisStore[7].Axis[1..15].Pos5.Speed := 0;
   AxisStore[8].Axis[1..15].Pos5.Speed := 0;
   AxisStore[9].Axis[1..15].Pos5.Speed := 0;
   AxisStore[10].Axis[1..15].Pos5.Speed := 0;
   AxisStore[11].Axis[1..15].Pos5.Speed := 0;
   AxisStore[12].Axis[1..15].Pos5.Speed := 0;
   AxisStore[13].Axis[1..15].Pos5.Speed := 0;
   AxisStore[14].Axis[1..15].Pos5.Speed := 0;
   AxisStore[15].Axis[1..15].Pos5.Speed := 0;
   AxisStore[1].Axis[1..15].Pos5.Reached := FALSE;
   AxisStore[2].Axis[1..15].Pos5.Reached := FALSE;
   AxisStore[3].Axis[1..15].Pos5.Reached := FALSE;
   AxisStore[4].Axis[1..15].Pos5.Reached := FALSE;
   AxisStore[5].Axis[1..15].Pos5.Reached := FALSE;
   AxisStore[6].Axis[1..15].Pos5.Reached := FALSE;
   AxisStore[7].Axis[1..15].Pos5.Reached := FALSE;
   AxisStore[8].Axis[1..15].Pos5.Reached := FALSE;
   AxisStore[9].Axis[1..15].Pos5.Reached := FALSE;
   AxisStore[10].Axis[1..15].Pos5.Reached := FALSE;
   AxisStore[11].Axis[1..15].Pos5.Reached := FALSE;
   AxisStore[12].Axis[1..15].Pos5.Reached := FALSE;
   AxisStore[13].Axis[1..15].Pos5.Reached := FALSE;
   AxisStore[14].Axis[1..15].Pos5.Reached := FALSE;
   AxisStore[15].Axis[1..15].Pos5.Reached := FALSE;
   AxisStore[1].Axis[1..15].Pos6.Position := 0.0;
   AxisStore[2].Axis[1..15].Pos6.Position := 0.0;
   AxisStore[3].Axis[1..15].Pos6.Position := 0.0;
   AxisStore[4].Axis[1..15].Pos6.Position := 0.0;
   AxisStore[5].Axis[1..15].Pos6.Position := 0.0;
   AxisStore[6].Axis[1..15].Pos6.Position := 0.0;
   AxisStore[7].Axis[1..15].Pos6.Position := 0.0;
   AxisStore[8].Axis[1..15].Pos6.Position := 0.0;
   AxisStore[9].Axis[1..15].Pos6.Position := 0.0;
   AxisStore[10].Axis[1..15].Pos6.Position := 0.0;
   AxisStore[11].Axis[1..15].Pos6.Position := 0.0;
   AxisStore[12].Axis[1..15].Pos6.Position := 0.0;
   AxisStore[13].Axis[1..15].Pos6.Position := 0.0;
   AxisStore[14].Axis[1..15].Pos6.Position := 0.0;
   AxisStore[15].Axis[1..15].Pos6.Position := 0.0;
   AxisStore[1].Axis[1..15].Pos6.Speed := 0;
   AxisStore[2].Axis[1..15].Pos6.Speed := 0;
   AxisStore[3].Axis[1..15].Pos6.Speed := 0;
   AxisStore[4].Axis[1..15].Pos6.Speed := 0;
   AxisStore[5].Axis[1..15].Pos6.Speed := 0;
   AxisStore[6].Axis[1..15].Pos6.Speed := 0;
   AxisStore[7].Axis[1..15].Pos6.Speed := 0;
   AxisStore[8].Axis[1..15].Pos6.Speed := 0;
   AxisStore[9].Axis[1..15].Pos6.Speed := 0;
   AxisStore[10].Axis[1..15].Pos6.Speed := 0;
   AxisStore[11].Axis[1..15].Pos6.Speed := 0;
   AxisStore[12].Axis[1..15].Pos6.Speed := 0;
   AxisStore[13].Axis[1..15].Pos6.Speed := 0;
   AxisStore[14].Axis[1..15].Pos6.Speed := 0;
   AxisStore[15].Axis[1..15].Pos6.Speed := 0;
   AxisStore[1].Axis[1..15].Pos6.Reached := FALSE;
   AxisStore[2].Axis[1..15].Pos6.Reached := FALSE;
   AxisStore[3].Axis[1..15].Pos6.Reached := FALSE;
   AxisStore[4].Axis[1..15].Pos6.Reached := FALSE;
   AxisStore[5].Axis[1..15].Pos6.Reached := FALSE;
   AxisStore[6].Axis[1..15].Pos6.Reached := FALSE;
   AxisStore[7].Axis[1..15].Pos6.Reached := FALSE;
   AxisStore[8].Axis[1..15].Pos6.Reached := FALSE;
   AxisStore[9].Axis[1..15].Pos6.Reached := FALSE;
   AxisStore[10].Axis[1..15].Pos6.Reached := FALSE;
   AxisStore[11].Axis[1..15].Pos6.Reached := FALSE;
   AxisStore[12].Axis[1..15].Pos6.Reached := FALSE;
   AxisStore[13].Axis[1..15].Pos6.Reached := FALSE;
   AxisStore[14].Axis[1..15].Pos6.Reached := FALSE;
   AxisStore[15].Axis[1..15].Pos6.Reached := FALSE;
   AxisStore[1].Axis[1..15].Pos7.Position := 0.0;
   AxisStore[2].Axis[1..15].Pos7.Position := 0.0;
   AxisStore[3].Axis[1..15].Pos7.Position := 0.0;
   AxisStore[4].Axis[1..15].Pos7.Position := 0.0;
   AxisStore[5].Axis[1..15].Pos7.Position := 0.0;
   AxisStore[6].Axis[1..15].Pos7.Position := 0.0;
   AxisStore[7].Axis[1..15].Pos7.Position := 0.0;
   AxisStore[8].Axis[1..15].Pos7.Position := 0.0;
   AxisStore[9].Axis[1..15].Pos7.Position := 0.0;
   AxisStore[10].Axis[1..15].Pos7.Position := 0.0;
   AxisStore[11].Axis[1..15].Pos7.Position := 0.0;
   AxisStore[12].Axis[1..15].Pos7.Position := 0.0;
   AxisStore[13].Axis[1..15].Pos7.Position := 0.0;
   AxisStore[14].Axis[1..15].Pos7.Position := 0.0;
   AxisStore[15].Axis[1..15].Pos7.Position := 0.0;
   AxisStore[1].Axis[1..15].Pos7.Speed := 0;
   AxisStore[2].Axis[1..15].Pos7.Speed := 0;
   AxisStore[3].Axis[1..15].Pos7.Speed := 0;
   AxisStore[4].Axis[1..15].Pos7.Speed := 0;
   AxisStore[5].Axis[1..15].Pos7.Speed := 0;
   AxisStore[6].Axis[1..15].Pos7.Speed := 0;
   AxisStore[7].Axis[1..15].Pos7.Speed := 0;
   AxisStore[8].Axis[1..15].Pos7.Speed := 0;
   AxisStore[9].Axis[1..15].Pos7.Speed := 0;
   AxisStore[10].Axis[1..15].Pos7.Speed := 0;
   AxisStore[11].Axis[1..15].Pos7.Speed := 0;
   AxisStore[12].Axis[1..15].Pos7.Speed := 0;
   AxisStore[13].Axis[1..15].Pos7.Speed := 0;
   AxisStore[14].Axis[1..15].Pos7.Speed := 0;
   AxisStore[15].Axis[1..15].Pos7.Speed := 0;
   AxisStore[1].Axis[1..15].Pos7.Reached := FALSE;
   AxisStore[2].Axis[1..15].Pos7.Reached := FALSE;
   AxisStore[3].Axis[1..15].Pos7.Reached := FALSE;
   AxisStore[4].Axis[1..15].Pos7.Reached := FALSE;
   AxisStore[5].Axis[1..15].Pos7.Reached := FALSE;
   AxisStore[6].Axis[1..15].Pos7.Reached := FALSE;
   AxisStore[7].Axis[1..15].Pos7.Reached := FALSE;
   AxisStore[8].Axis[1..15].Pos7.Reached := FALSE;
   AxisStore[9].Axis[1..15].Pos7.Reached := FALSE;
   AxisStore[10].Axis[1..15].Pos7.Reached := FALSE;
   AxisStore[11].Axis[1..15].Pos7.Reached := FALSE;
   AxisStore[12].Axis[1..15].Pos7.Reached := FALSE;
   AxisStore[13].Axis[1..15].Pos7.Reached := FALSE;
   AxisStore[14].Axis[1..15].Pos7.Reached := FALSE;
   AxisStore[15].Axis[1..15].Pos7.Reached := FALSE;
   AxisStore[1].Axis[1..15].Pos8.Position := 0.0;
   AxisStore[2].Axis[1..15].Pos8.Position := 0.0;
   AxisStore[3].Axis[1..15].Pos8.Position := 0.0;
   AxisStore[4].Axis[1..15].Pos8.Position := 0.0;
   AxisStore[5].Axis[1..15].Pos8.Position := 0.0;
   AxisStore[6].Axis[1..15].Pos8.Position := 0.0;
   AxisStore[7].Axis[1..15].Pos8.Position := 0.0;
   AxisStore[8].Axis[1..15].Pos8.Position := 0.0;
   AxisStore[9].Axis[1..15].Pos8.Position := 0.0;
   AxisStore[10].Axis[1..15].Pos8.Position := 0.0;
   AxisStore[11].Axis[1..15].Pos8.Position := 0.0;
   AxisStore[12].Axis[1..15].Pos8.Position := 0.0;
   AxisStore[13].Axis[1..15].Pos8.Position := 0.0;
   AxisStore[14].Axis[1..15].Pos8.Position := 0.0;
   AxisStore[15].Axis[1..15].Pos8.Position := 0.0;
   AxisStore[1].Axis[1..15].Pos8.Speed := 0;
   AxisStore[2].Axis[1..15].Pos8.Speed := 0;
   AxisStore[3].Axis[1..15].Pos8.Speed := 0;
   AxisStore[4].Axis[1..15].Pos8.Speed := 0;
   AxisStore[5].Axis[1..15].Pos8.Speed := 0;
   AxisStore[6].Axis[1..15].Pos8.Speed := 0;
   AxisStore[7].Axis[1..15].Pos8.Speed := 0;
   AxisStore[8].Axis[1..15].Pos8.Speed := 0;
   AxisStore[9].Axis[1..15].Pos8.Speed := 0;
   AxisStore[10].Axis[1..15].Pos8.Speed := 0;
   AxisStore[11].Axis[1..15].Pos8.Speed := 0;
   AxisStore[12].Axis[1..15].Pos8.Speed := 0;
   AxisStore[13].Axis[1..15].Pos8.Speed := 0;
   AxisStore[14].Axis[1..15].Pos8.Speed := 0;
   AxisStore[15].Axis[1..15].Pos8.Speed := 0;
   AxisStore[1].Axis[1..15].Pos8.Reached := FALSE;
   AxisStore[2].Axis[1..15].Pos8.Reached := FALSE;
   AxisStore[3].Axis[1..15].Pos8.Reached := FALSE;
   AxisStore[4].Axis[1..15].Pos8.Reached := FALSE;
   AxisStore[5].Axis[1..15].Pos8.Reached := FALSE;
   AxisStore[6].Axis[1..15].Pos8.Reached := FALSE;
   AxisStore[7].Axis[1..15].Pos8.Reached := FALSE;
   AxisStore[8].Axis[1..15].Pos8.Reached := FALSE;
   AxisStore[9].Axis[1..15].Pos8.Reached := FALSE;
   AxisStore[10].Axis[1..15].Pos8.Reached := FALSE;
   AxisStore[11].Axis[1..15].Pos8.Reached := FALSE;
   AxisStore[12].Axis[1..15].Pos8.Reached := FALSE;
   AxisStore[13].Axis[1..15].Pos8.Reached := FALSE;
   AxisStore[14].Axis[1..15].Pos8.Reached := FALSE;
   AxisStore[15].Axis[1..15].Pos8.Reached := FALSE;
   AxisStore[1].Axis[1..15].Pos9.Position := 0.0;
   AxisStore[2].Axis[1..15].Pos9.Position := 0.0;
   AxisStore[3].Axis[1..15].Pos9.Position := 0.0;
   AxisStore[4].Axis[1..15].Pos9.Position := 0.0;
   AxisStore[5].Axis[1..15].Pos9.Position := 0.0;
   AxisStore[6].Axis[1..15].Pos9.Position := 0.0;
   AxisStore[7].Axis[1..15].Pos9.Position := 0.0;
   AxisStore[8].Axis[1..15].Pos9.Position := 0.0;
   AxisStore[9].Axis[1..15].Pos9.Position := 0.0;
   AxisStore[10].Axis[1..15].Pos9.Position := 0.0;
   AxisStore[11].Axis[1..15].Pos9.Position := 0.0;
   AxisStore[12].Axis[1..15].Pos9.Position := 0.0;
   AxisStore[13].Axis[1..15].Pos9.Position := 0.0;
   AxisStore[14].Axis[1..15].Pos9.Position := 0.0;
   AxisStore[15].Axis[1..15].Pos9.Position := 0.0;
   AxisStore[1].Axis[1..15].Pos9.Speed := 0;
   AxisStore[2].Axis[1..15].Pos9.Speed := 0;
   AxisStore[3].Axis[1..15].Pos9.Speed := 0;
   AxisStore[4].Axis[1..15].Pos9.Speed := 0;
   AxisStore[5].Axis[1..15].Pos9.Speed := 0;
   AxisStore[6].Axis[1..15].Pos9.Speed := 0;
   AxisStore[7].Axis[1..15].Pos9.Speed := 0;
   AxisStore[8].Axis[1..15].Pos9.Speed := 0;
   AxisStore[9].Axis[1..15].Pos9.Speed := 0;
   AxisStore[10].Axis[1..15].Pos9.Speed := 0;
   AxisStore[11].Axis[1..15].Pos9.Speed := 0;
   AxisStore[12].Axis[1..15].Pos9.Speed := 0;
   AxisStore[13].Axis[1..15].Pos9.Speed := 0;
   AxisStore[14].Axis[1..15].Pos9.Speed := 0;
   AxisStore[15].Axis[1..15].Pos9.Speed := 0;
   AxisStore[1].Axis[1..15].Pos9.Reached := FALSE;
   AxisStore[2].Axis[1..15].Pos9.Reached := FALSE;
   AxisStore[3].Axis[1..15].Pos9.Reached := FALSE;
   AxisStore[4].Axis[1..15].Pos9.Reached := FALSE;
   AxisStore[5].Axis[1..15].Pos9.Reached := FALSE;
   AxisStore[6].Axis[1..15].Pos9.Reached := FALSE;
   AxisStore[7].Axis[1..15].Pos9.Reached := FALSE;
   AxisStore[8].Axis[1..15].Pos9.Reached := FALSE;
   AxisStore[9].Axis[1..15].Pos9.Reached := FALSE;
   AxisStore[10].Axis[1..15].Pos9.Reached := FALSE;
   AxisStore[11].Axis[1..15].Pos9.Reached := FALSE;
   AxisStore[12].Axis[1..15].Pos9.Reached := FALSE;
   AxisStore[13].Axis[1..15].Pos9.Reached := FALSE;
   AxisStore[14].Axis[1..15].Pos9.Reached := FALSE;
   AxisStore[15].Axis[1..15].Pos9.Reached := FALSE;
   AxisStore[1].Axis[1..15].Pos10.Position := 0.0;
   AxisStore[2].Axis[1..15].Pos10.Position := 0.0;
   AxisStore[3].Axis[1..15].Pos10.Position := 0.0;
   AxisStore[4].Axis[1..15].Pos10.Position := 0.0;
   AxisStore[5].Axis[1..15].Pos10.Position := 0.0;
   AxisStore[6].Axis[1..15].Pos10.Position := 0.0;
   AxisStore[7].Axis[1..15].Pos10.Position := 0.0;
   AxisStore[8].Axis[1..15].Pos10.Position := 0.0;
   AxisStore[9].Axis[1..15].Pos10.Position := 0.0;
   AxisStore[10].Axis[1..15].Pos10.Position := 0.0;
   AxisStore[11].Axis[1..15].Pos10.Position := 0.0;
   AxisStore[12].Axis[1..15].Pos10.Position := 0.0;
   AxisStore[13].Axis[1..15].Pos10.Position := 0.0;
   AxisStore[14].Axis[1..15].Pos10.Position := 0.0;
   AxisStore[15].Axis[1..15].Pos10.Position := 0.0;
   AxisStore[1].Axis[1..15].Pos10.Speed := 0;
   AxisStore[2].Axis[1..15].Pos10.Speed := 0;
   AxisStore[3].Axis[1..15].Pos10.Speed := 0;
   AxisStore[4].Axis[1..15].Pos10.Speed := 0;
   AxisStore[5].Axis[1..15].Pos10.Speed := 0;
   AxisStore[6].Axis[1..15].Pos10.Speed := 0;
   AxisStore[7].Axis[1..15].Pos10.Speed := 0;
   AxisStore[8].Axis[1..15].Pos10.Speed := 0;
   AxisStore[9].Axis[1..15].Pos10.Speed := 0;
   AxisStore[10].Axis[1..15].Pos10.Speed := 0;
   AxisStore[11].Axis[1..15].Pos10.Speed := 0;
   AxisStore[12].Axis[1..15].Pos10.Speed := 0;
   AxisStore[13].Axis[1..15].Pos10.Speed := 0;
   AxisStore[14].Axis[1..15].Pos10.Speed := 0;
   AxisStore[15].Axis[1..15].Pos10.Speed := 0;
   AxisStore[1].Axis[1..15].Pos10.Reached := FALSE;
   AxisStore[2].Axis[1..15].Pos10.Reached := FALSE;
   AxisStore[3].Axis[1..15].Pos10.Reached := FALSE;
   AxisStore[4].Axis[1..15].Pos10.Reached := FALSE;
   AxisStore[5].Axis[1..15].Pos10.Reached := FALSE;
   AxisStore[6].Axis[1..15].Pos10.Reached := FALSE;
   AxisStore[7].Axis[1..15].Pos10.Reached := FALSE;
   AxisStore[8].Axis[1..15].Pos10.Reached := FALSE;
   AxisStore[9].Axis[1..15].Pos10.Reached := FALSE;
   AxisStore[10].Axis[1..15].Pos10.Reached := FALSE;
   AxisStore[11].Axis[1..15].Pos10.Reached := FALSE;
   AxisStore[12].Axis[1..15].Pos10.Reached := FALSE;
   AxisStore[13].Axis[1..15].Pos10.Reached := FALSE;
   AxisStore[14].Axis[1..15].Pos10.Reached := FALSE;
   AxisStore[15].Axis[1..15].Pos10.Reached := FALSE;
   AxisStore[1].Axis[1..15].Pos11.Position := 0.0;
   AxisStore[2].Axis[1..15].Pos11.Position := 0.0;
   AxisStore[3].Axis[1..15].Pos11.Position := 0.0;
   AxisStore[4].Axis[1..15].Pos11.Position := 0.0;
   AxisStore[5].Axis[1..15].Pos11.Position := 0.0;
   AxisStore[6].Axis[1..15].Pos11.Position := 0.0;
   AxisStore[7].Axis[1..15].Pos11.Position := 0.0;
   AxisStore[8].Axis[1..15].Pos11.Position := 0.0;
   AxisStore[9].Axis[1..15].Pos11.Position := 0.0;
   AxisStore[10].Axis[1..15].Pos11.Position := 0.0;
   AxisStore[11].Axis[1..15].Pos11.Position := 0.0;
   AxisStore[12].Axis[1..15].Pos11.Position := 0.0;
   AxisStore[13].Axis[1..15].Pos11.Position := 0.0;
   AxisStore[14].Axis[1..15].Pos11.Position := 0.0;
   AxisStore[15].Axis[1..15].Pos11.Position := 0.0;
   AxisStore[1].Axis[1..15].Pos11.Speed := 0;
   AxisStore[2].Axis[1..15].Pos11.Speed := 0;
   AxisStore[3].Axis[1..15].Pos11.Speed := 0;
   AxisStore[4].Axis[1..15].Pos11.Speed := 0;
   AxisStore[5].Axis[1..15].Pos11.Speed := 0;
   AxisStore[6].Axis[1..15].Pos11.Speed := 0;
   AxisStore[7].Axis[1..15].Pos11.Speed := 0;
   AxisStore[8].Axis[1..15].Pos11.Speed := 0;
   AxisStore[9].Axis[1..15].Pos11.Speed := 0;
   AxisStore[10].Axis[1..15].Pos11.Speed := 0;
   AxisStore[11].Axis[1..15].Pos11.Speed := 0;
   AxisStore[12].Axis[1..15].Pos11.Speed := 0;
   AxisStore[13].Axis[1..15].Pos11.Speed := 0;
   AxisStore[14].Axis[1..15].Pos11.Speed := 0;
   AxisStore[15].Axis[1..15].Pos11.Speed := 0;
   AxisStore[1].Axis[1..15].Pos11.Reached := FALSE;
   AxisStore[2].Axis[1..15].Pos11.Reached := FALSE;
   AxisStore[3].Axis[1..15].Pos11.Reached := FALSE;
   AxisStore[4].Axis[1..15].Pos11.Reached := FALSE;
   AxisStore[5].Axis[1..15].Pos11.Reached := FALSE;
   AxisStore[6].Axis[1..15].Pos11.Reached := FALSE;
   AxisStore[7].Axis[1..15].Pos11.Reached := FALSE;
   AxisStore[8].Axis[1..15].Pos11.Reached := FALSE;
   AxisStore[9].Axis[1..15].Pos11.Reached := FALSE;
   AxisStore[10].Axis[1..15].Pos11.Reached := FALSE;
   AxisStore[11].Axis[1..15].Pos11.Reached := FALSE;
   AxisStore[12].Axis[1..15].Pos11.Reached := FALSE;
   AxisStore[13].Axis[1..15].Pos11.Reached := FALSE;
   AxisStore[14].Axis[1..15].Pos11.Reached := FALSE;
   AxisStore[15].Axis[1..15].Pos11.Reached := FALSE;
   AxisStore[1].Axis[1..15].Pos12.Position := 0.0;
   AxisStore[2].Axis[1..15].Pos12.Position := 0.0;
   AxisStore[3].Axis[1..15].Pos12.Position := 0.0;
   AxisStore[4].Axis[1..15].Pos12.Position := 0.0;
   AxisStore[5].Axis[1..15].Pos12.Position := 0.0;
   AxisStore[6].Axis[1..15].Pos12.Position := 0.0;
   AxisStore[7].Axis[1..15].Pos12.Position := 0.0;
   AxisStore[8].Axis[1..15].Pos12.Position := 0.0;
   AxisStore[9].Axis[1..15].Pos12.Position := 0.0;
   AxisStore[10].Axis[1..15].Pos12.Position := 0.0;
   AxisStore[11].Axis[1..15].Pos12.Position := 0.0;
   AxisStore[12].Axis[1..15].Pos12.Position := 0.0;
   AxisStore[13].Axis[1..15].Pos12.Position := 0.0;
   AxisStore[14].Axis[1..15].Pos12.Position := 0.0;
   AxisStore[15].Axis[1..15].Pos12.Position := 0.0;
   AxisStore[1].Axis[1..15].Pos12.Speed := 0;
   AxisStore[2].Axis[1..15].Pos12.Speed := 0;
   AxisStore[3].Axis[1..15].Pos12.Speed := 0;
   AxisStore[4].Axis[1..15].Pos12.Speed := 0;
   AxisStore[5].Axis[1..15].Pos12.Speed := 0;
   AxisStore[6].Axis[1..15].Pos12.Speed := 0;
   AxisStore[7].Axis[1..15].Pos12.Speed := 0;
   AxisStore[8].Axis[1..15].Pos12.Speed := 0;
   AxisStore[9].Axis[1..15].Pos12.Speed := 0;
   AxisStore[10].Axis[1..15].Pos12.Speed := 0;
   AxisStore[11].Axis[1..15].Pos12.Speed := 0;
   AxisStore[12].Axis[1..15].Pos12.Speed := 0;
   AxisStore[13].Axis[1..15].Pos12.Speed := 0;
   AxisStore[14].Axis[1..15].Pos12.Speed := 0;
   AxisStore[15].Axis[1..15].Pos12.Speed := 0;
   AxisStore[1].Axis[1..15].Pos12.Reached := FALSE;
   AxisStore[2].Axis[1..15].Pos12.Reached := FALSE;
   AxisStore[3].Axis[1..15].Pos12.Reached := FALSE;
   AxisStore[4].Axis[1..15].Pos12.Reached := FALSE;
   AxisStore[5].Axis[1..15].Pos12.Reached := FALSE;
   AxisStore[6].Axis[1..15].Pos12.Reached := FALSE;
   AxisStore[7].Axis[1..15].Pos12.Reached := FALSE;
   AxisStore[8].Axis[1..15].Pos12.Reached := FALSE;
   AxisStore[9].Axis[1..15].Pos12.Reached := FALSE;
   AxisStore[10].Axis[1..15].Pos12.Reached := FALSE;
   AxisStore[11].Axis[1..15].Pos12.Reached := FALSE;
   AxisStore[12].Axis[1..15].Pos12.Reached := FALSE;
   AxisStore[13].Axis[1..15].Pos12.Reached := FALSE;
   AxisStore[14].Axis[1..15].Pos12.Reached := FALSE;
   AxisStore[15].Axis[1..15].Pos12.Reached := FALSE;
   AxisStore[1].Axis[1..15].Pos13.Position := 0.0;
   AxisStore[2].Axis[1..15].Pos13.Position := 0.0;
   AxisStore[3].Axis[1..15].Pos13.Position := 0.0;
   AxisStore[4].Axis[1..15].Pos13.Position := 0.0;
   AxisStore[5].Axis[1..15].Pos13.Position := 0.0;
   AxisStore[6].Axis[1..15].Pos13.Position := 0.0;
   AxisStore[7].Axis[1..15].Pos13.Position := 0.0;
   AxisStore[8].Axis[1..15].Pos13.Position := 0.0;
   AxisStore[9].Axis[1..15].Pos13.Position := 0.0;
   AxisStore[10].Axis[1..15].Pos13.Position := 0.0;
   AxisStore[11].Axis[1..15].Pos13.Position := 0.0;
   AxisStore[12].Axis[1..15].Pos13.Position := 0.0;
   AxisStore[13].Axis[1..15].Pos13.Position := 0.0;
   AxisStore[14].Axis[1..15].Pos13.Position := 0.0;
   AxisStore[15].Axis[1..15].Pos13.Position := 0.0;
   AxisStore[1].Axis[1..15].Pos13.Speed := 0;
   AxisStore[2].Axis[1..15].Pos13.Speed := 0;
   AxisStore[3].Axis[1..15].Pos13.Speed := 0;
   AxisStore[4].Axis[1..15].Pos13.Speed := 0;
   AxisStore[5].Axis[1..15].Pos13.Speed := 0;
   AxisStore[6].Axis[1..15].Pos13.Speed := 0;
   AxisStore[7].Axis[1..15].Pos13.Speed := 0;
   AxisStore[8].Axis[1..15].Pos13.Speed := 0;
   AxisStore[9].Axis[1..15].Pos13.Speed := 0;
   AxisStore[10].Axis[1..15].Pos13.Speed := 0;
   AxisStore[11].Axis[1..15].Pos13.Speed := 0;
   AxisStore[12].Axis[1..15].Pos13.Speed := 0;
   AxisStore[13].Axis[1..15].Pos13.Speed := 0;
   AxisStore[14].Axis[1..15].Pos13.Speed := 0;
   AxisStore[15].Axis[1..15].Pos13.Speed := 0;
   AxisStore[1].Axis[1..15].Pos13.Reached := FALSE;
   AxisStore[2].Axis[1..15].Pos13.Reached := FALSE;
   AxisStore[3].Axis[1..15].Pos13.Reached := FALSE;
   AxisStore[4].Axis[1..15].Pos13.Reached := FALSE;
   AxisStore[5].Axis[1..15].Pos13.Reached := FALSE;
   AxisStore[6].Axis[1..15].Pos13.Reached := FALSE;
   AxisStore[7].Axis[1..15].Pos13.Reached := FALSE;
   AxisStore[8].Axis[1..15].Pos13.Reached := FALSE;
   AxisStore[9].Axis[1..15].Pos13.Reached := FALSE;
   AxisStore[10].Axis[1..15].Pos13.Reached := FALSE;
   AxisStore[11].Axis[1..15].Pos13.Reached := FALSE;
   AxisStore[12].Axis[1..15].Pos13.Reached := FALSE;
   AxisStore[13].Axis[1..15].Pos13.Reached := FALSE;
   AxisStore[14].Axis[1..15].Pos13.Reached := FALSE;
   AxisStore[15].Axis[1..15].Pos13.Reached := FALSE;
   AxisStore[1].Axis[1..15].Pos14.Position := 0.0;
   AxisStore[2].Axis[1..15].Pos14.Position := 0.0;
   AxisStore[3].Axis[1..15].Pos14.Position := 0.0;
   AxisStore[4].Axis[1..15].Pos14.Position := 0.0;
   AxisStore[5].Axis[1..15].Pos14.Position := 0.0;
   AxisStore[6].Axis[1..15].Pos14.Position := 0.0;
   AxisStore[7].Axis[1..15].Pos14.Position := 0.0;
   AxisStore[8].Axis[1..15].Pos14.Position := 0.0;
   AxisStore[9].Axis[1..15].Pos14.Position := 0.0;
   AxisStore[10].Axis[1..15].Pos14.Position := 0.0;
   AxisStore[11].Axis[1..15].Pos14.Position := 0.0;
   AxisStore[12].Axis[1..15].Pos14.Position := 0.0;
   AxisStore[13].Axis[1..15].Pos14.Position := 0.0;
   AxisStore[14].Axis[1..15].Pos14.Position := 0.0;
   AxisStore[15].Axis[1..15].Pos14.Position := 0.0;
   AxisStore[1].Axis[1..15].Pos14.Speed := 0;
   AxisStore[2].Axis[1..15].Pos14.Speed := 0;
   AxisStore[3].Axis[1..15].Pos14.Speed := 0;
   AxisStore[4].Axis[1..15].Pos14.Speed := 0;
   AxisStore[5].Axis[1..15].Pos14.Speed := 0;
   AxisStore[6].Axis[1..15].Pos14.Speed := 0;
   AxisStore[7].Axis[1..15].Pos14.Speed := 0;
   AxisStore[8].Axis[1..15].Pos14.Speed := 0;
   AxisStore[9].Axis[1..15].Pos14.Speed := 0;
   AxisStore[10].Axis[1..15].Pos14.Speed := 0;
   AxisStore[11].Axis[1..15].Pos14.Speed := 0;
   AxisStore[12].Axis[1..15].Pos14.Speed := 0;
   AxisStore[13].Axis[1..15].Pos14.Speed := 0;
   AxisStore[14].Axis[1..15].Pos14.Speed := 0;
   AxisStore[15].Axis[1..15].Pos14.Speed := 0;
   AxisStore[1].Axis[1..15].Pos14.Reached := FALSE;
   AxisStore[2].Axis[1..15].Pos14.Reached := FALSE;
   AxisStore[3].Axis[1..15].Pos14.Reached := FALSE;
   AxisStore[4].Axis[1..15].Pos14.Reached := FALSE;
   AxisStore[5].Axis[1..15].Pos14.Reached := FALSE;
   AxisStore[6].Axis[1..15].Pos14.Reached := FALSE;
   AxisStore[7].Axis[1..15].Pos14.Reached := FALSE;
   AxisStore[8].Axis[1..15].Pos14.Reached := FALSE;
   AxisStore[9].Axis[1..15].Pos14.Reached := FALSE;
   AxisStore[10].Axis[1..15].Pos14.Reached := FALSE;
   AxisStore[11].Axis[1..15].Pos14.Reached := FALSE;
   AxisStore[12].Axis[1..15].Pos14.Reached := FALSE;
   AxisStore[13].Axis[1..15].Pos14.Reached := FALSE;
   AxisStore[14].Axis[1..15].Pos14.Reached := FALSE;
   AxisStore[15].Axis[1..15].Pos14.Reached := FALSE;
   AxisStore[1].Axis[1..15].Pos15.Position := 0.0;
   AxisStore[2].Axis[1..15].Pos15.Position := 0.0;
   AxisStore[3].Axis[1..15].Pos15.Position := 0.0;
   AxisStore[4].Axis[1..15].Pos15.Position := 0.0;
   AxisStore[5].Axis[1..15].Pos15.Position := 0.0;
   AxisStore[6].Axis[1..15].Pos15.Position := 0.0;
   AxisStore[7].Axis[1..15].Pos15.Position := 0.0;
   AxisStore[8].Axis[1..15].Pos15.Position := 0.0;
   AxisStore[9].Axis[1..15].Pos15.Position := 0.0;
   AxisStore[10].Axis[1..15].Pos15.Position := 0.0;
   AxisStore[11].Axis[1..15].Pos15.Position := 0.0;
   AxisStore[12].Axis[1..15].Pos15.Position := 0.0;
   AxisStore[13].Axis[1..15].Pos15.Position := 0.0;
   AxisStore[14].Axis[1..15].Pos15.Position := 0.0;
   AxisStore[15].Axis[1..15].Pos15.Position := 0.0;
   AxisStore[1].Axis[1..15].Pos15.Speed := 0;
   AxisStore[2].Axis[1..15].Pos15.Speed := 0;
   AxisStore[3].Axis[1..15].Pos15.Speed := 0;
   AxisStore[4].Axis[1..15].Pos15.Speed := 0;
   AxisStore[5].Axis[1..15].Pos15.Speed := 0;
   AxisStore[6].Axis[1..15].Pos15.Speed := 0;
   AxisStore[7].Axis[1..15].Pos15.Speed := 0;
   AxisStore[8].Axis[1..15].Pos15.Speed := 0;
   AxisStore[9].Axis[1..15].Pos15.Speed := 0;
   AxisStore[10].Axis[1..15].Pos15.Speed := 0;
   AxisStore[11].Axis[1..15].Pos15.Speed := 0;
   AxisStore[12].Axis[1..15].Pos15.Speed := 0;
   AxisStore[13].Axis[1..15].Pos15.Speed := 0;
   AxisStore[14].Axis[1..15].Pos15.Speed := 0;
   AxisStore[15].Axis[1..15].Pos15.Speed := 0;
   AxisStore[1].Axis[1..15].Pos15.Reached := FALSE;
   AxisStore[2].Axis[1..15].Pos15.Reached := FALSE;
   AxisStore[3].Axis[1..15].Pos15.Reached := FALSE;
   AxisStore[4].Axis[1..15].Pos15.Reached := FALSE;
   AxisStore[5].Axis[1..15].Pos15.Reached := FALSE;
   AxisStore[6].Axis[1..15].Pos15.Reached := FALSE;
   AxisStore[7].Axis[1..15].Pos15.Reached := FALSE;
   AxisStore[8].Axis[1..15].Pos15.Reached := FALSE;
   AxisStore[9].Axis[1..15].Pos15.Reached := FALSE;
   AxisStore[10].Axis[1..15].Pos15.Reached := FALSE;
   AxisStore[11].Axis[1..15].Pos15.Reached := FALSE;
   AxisStore[12].Axis[1..15].Pos15.Reached := FALSE;
   AxisStore[13].Axis[1..15].Pos15.Reached := FALSE;
   AxisStore[14].Axis[1..15].Pos15.Reached := FALSE;
   AxisStore[15].Axis[1..15].Pos15.Reached := FALSE;
   AxisStore[1].Axis[1..15].Pos16.Position := 0.0;
   AxisStore[2].Axis[1..15].Pos16.Position := 0.0;
   AxisStore[3].Axis[1..15].Pos16.Position := 0.0;
   AxisStore[4].Axis[1..15].Pos16.Position := 0.0;
   AxisStore[5].Axis[1..15].Pos16.Position := 0.0;
   AxisStore[6].Axis[1..15].Pos16.Position := 0.0;
   AxisStore[7].Axis[1..15].Pos16.Position := 0.0;
   AxisStore[8].Axis[1..15].Pos16.Position := 0.0;
   AxisStore[9].Axis[1..15].Pos16.Position := 0.0;
   AxisStore[10].Axis[1..15].Pos16.Position := 0.0;
   AxisStore[11].Axis[1..15].Pos16.Position := 0.0;
   AxisStore[12].Axis[1..15].Pos16.Position := 0.0;
   AxisStore[13].Axis[1..15].Pos16.Position := 0.0;
   AxisStore[14].Axis[1..15].Pos16.Position := 0.0;
   AxisStore[15].Axis[1..15].Pos16.Position := 0.0;
   AxisStore[1].Axis[1..15].Pos16.Speed := 0;
   AxisStore[2].Axis[1..15].Pos16.Speed := 0;
   AxisStore[3].Axis[1..15].Pos16.Speed := 0;
   AxisStore[4].Axis[1..15].Pos16.Speed := 0;
   AxisStore[5].Axis[1..15].Pos16.Speed := 0;
   AxisStore[6].Axis[1..15].Pos16.Speed := 0;
   AxisStore[7].Axis[1..15].Pos16.Speed := 0;
   AxisStore[8].Axis[1..15].Pos16.Speed := 0;
   AxisStore[9].Axis[1..15].Pos16.Speed := 0;
   AxisStore[10].Axis[1..15].Pos16.Speed := 0;
   AxisStore[11].Axis[1..15].Pos16.Speed := 0;
   AxisStore[12].Axis[1..15].Pos16.Speed := 0;
   AxisStore[13].Axis[1..15].Pos16.Speed := 0;
   AxisStore[14].Axis[1..15].Pos16.Speed := 0;
   AxisStore[15].Axis[1..15].Pos16.Speed := 0;
   AxisStore[1].Axis[1..15].Pos16.Reached := FALSE;
   AxisStore[2].Axis[1..15].Pos16.Reached := FALSE;
   AxisStore[3].Axis[1..15].Pos16.Reached := FALSE;
   AxisStore[4].Axis[1..15].Pos16.Reached := FALSE;
   AxisStore[5].Axis[1..15].Pos16.Reached := FALSE;
   AxisStore[6].Axis[1..15].Pos16.Reached := FALSE;
   AxisStore[7].Axis[1..15].Pos16.Reached := FALSE;
   AxisStore[8].Axis[1..15].Pos16.Reached := FALSE;
   AxisStore[9].Axis[1..15].Pos16.Reached := FALSE;
   AxisStore[10].Axis[1..15].Pos16.Reached := FALSE;
   AxisStore[11].Axis[1..15].Pos16.Reached := FALSE;
   AxisStore[12].Axis[1..15].Pos16.Reached := FALSE;
   AxisStore[13].Axis[1..15].Pos16.Reached := FALSE;
   AxisStore[14].Axis[1..15].Pos16.Reached := FALSE;
   AxisStore[15].Axis[1..15].Pos16.Reached := FALSE;
   AxisStore[1].Axis[1..15].Pos17.Position := 0.0;
   AxisStore[2].Axis[1..15].Pos17.Position := 0.0;
   AxisStore[3].Axis[1..15].Pos17.Position := 0.0;
   AxisStore[4].Axis[1..15].Pos17.Position := 0.0;
   AxisStore[5].Axis[1..15].Pos17.Position := 0.0;
   AxisStore[6].Axis[1..15].Pos17.Position := 0.0;
   AxisStore[7].Axis[1..15].Pos17.Position := 0.0;
   AxisStore[8].Axis[1..15].Pos17.Position := 0.0;
   AxisStore[9].Axis[1..15].Pos17.Position := 0.0;
   AxisStore[10].Axis[1..15].Pos17.Position := 0.0;
   AxisStore[11].Axis[1..15].Pos17.Position := 0.0;
   AxisStore[12].Axis[1..15].Pos17.Position := 0.0;
   AxisStore[13].Axis[1..15].Pos17.Position := 0.0;
   AxisStore[14].Axis[1..15].Pos17.Position := 0.0;
   AxisStore[15].Axis[1..15].Pos17.Position := 0.0;
   AxisStore[1].Axis[1..15].Pos17.Speed := 0;
   AxisStore[2].Axis[1..15].Pos17.Speed := 0;
   AxisStore[3].Axis[1..15].Pos17.Speed := 0;
   AxisStore[4].Axis[1..15].Pos17.Speed := 0;
   AxisStore[5].Axis[1..15].Pos17.Speed := 0;
   AxisStore[6].Axis[1..15].Pos17.Speed := 0;
   AxisStore[7].Axis[1..15].Pos17.Speed := 0;
   AxisStore[8].Axis[1..15].Pos17.Speed := 0;
   AxisStore[9].Axis[1..15].Pos17.Speed := 0;
   AxisStore[10].Axis[1..15].Pos17.Speed := 0;
   AxisStore[11].Axis[1..15].Pos17.Speed := 0;
   AxisStore[12].Axis[1..15].Pos17.Speed := 0;
   AxisStore[13].Axis[1..15].Pos17.Speed := 0;
   AxisStore[14].Axis[1..15].Pos17.Speed := 0;
   AxisStore[15].Axis[1..15].Pos17.Speed := 0;
   AxisStore[1].Axis[1..15].Pos17.Reached := FALSE;
   AxisStore[2].Axis[1..15].Pos17.Reached := FALSE;
   AxisStore[3].Axis[1..15].Pos17.Reached := FALSE;
   AxisStore[4].Axis[1..15].Pos17.Reached := FALSE;
   AxisStore[5].Axis[1..15].Pos17.Reached := FALSE;
   AxisStore[6].Axis[1..15].Pos17.Reached := FALSE;
   AxisStore[7].Axis[1..15].Pos17.Reached := FALSE;
   AxisStore[8].Axis[1..15].Pos17.Reached := FALSE;
   AxisStore[9].Axis[1..15].Pos17.Reached := FALSE;
   AxisStore[10].Axis[1..15].Pos17.Reached := FALSE;
   AxisStore[11].Axis[1..15].Pos17.Reached := FALSE;
   AxisStore[12].Axis[1..15].Pos17.Reached := FALSE;
   AxisStore[13].Axis[1..15].Pos17.Reached := FALSE;
   AxisStore[14].Axis[1..15].Pos17.Reached := FALSE;
   AxisStore[15].Axis[1..15].Pos17.Reached := FALSE;
   AxisStore[1].Axis[1..15].Pos18.Position := 0.0;
   AxisStore[2].Axis[1..15].Pos18.Position := 0.0;
   AxisStore[3].Axis[1..15].Pos18.Position := 0.0;
   AxisStore[4].Axis[1..15].Pos18.Position := 0.0;
   AxisStore[5].Axis[1..15].Pos18.Position := 0.0;
   AxisStore[6].Axis[1..15].Pos18.Position := 0.0;
   AxisStore[7].Axis[1..15].Pos18.Position := 0.0;
   AxisStore[8].Axis[1..15].Pos18.Position := 0.0;
   AxisStore[9].Axis[1..15].Pos18.Position := 0.0;
   AxisStore[10].Axis[1..15].Pos18.Position := 0.0;
   AxisStore[11].Axis[1..15].Pos18.Position := 0.0;
   AxisStore[12].Axis[1..15].Pos18.Position := 0.0;
   AxisStore[13].Axis[1..15].Pos18.Position := 0.0;
   AxisStore[14].Axis[1..15].Pos18.Position := 0.0;
   AxisStore[15].Axis[1..15].Pos18.Position := 0.0;
   AxisStore[1].Axis[1..15].Pos18.Speed := 0;
   AxisStore[2].Axis[1..15].Pos18.Speed := 0;
   AxisStore[3].Axis[1..15].Pos18.Speed := 0;
   AxisStore[4].Axis[1..15].Pos18.Speed := 0;
   AxisStore[5].Axis[1..15].Pos18.Speed := 0;
   AxisStore[6].Axis[1..15].Pos18.Speed := 0;
   AxisStore[7].Axis[1..15].Pos18.Speed := 0;
   AxisStore[8].Axis[1..15].Pos18.Speed := 0;
   AxisStore[9].Axis[1..15].Pos18.Speed := 0;
   AxisStore[10].Axis[1..15].Pos18.Speed := 0;
   AxisStore[11].Axis[1..15].Pos18.Speed := 0;
   AxisStore[12].Axis[1..15].Pos18.Speed := 0;
   AxisStore[13].Axis[1..15].Pos18.Speed := 0;
   AxisStore[14].Axis[1..15].Pos18.Speed := 0;
   AxisStore[15].Axis[1..15].Pos18.Speed := 0;
   AxisStore[1].Axis[1..15].Pos18.Reached := FALSE;
   AxisStore[2].Axis[1..15].Pos18.Reached := FALSE;
   AxisStore[3].Axis[1..15].Pos18.Reached := FALSE;
   AxisStore[4].Axis[1..15].Pos18.Reached := FALSE;
   AxisStore[5].Axis[1..15].Pos18.Reached := FALSE;
   AxisStore[6].Axis[1..15].Pos18.Reached := FALSE;
   AxisStore[7].Axis[1..15].Pos18.Reached := FALSE;
   AxisStore[8].Axis[1..15].Pos18.Reached := FALSE;
   AxisStore[9].Axis[1..15].Pos18.Reached := FALSE;
   AxisStore[10].Axis[1..15].Pos18.Reached := FALSE;
   AxisStore[11].Axis[1..15].Pos18.Reached := FALSE;
   AxisStore[12].Axis[1..15].Pos18.Reached := FALSE;
   AxisStore[13].Axis[1..15].Pos18.Reached := FALSE;
   AxisStore[14].Axis[1..15].Pos18.Reached := FALSE;
   AxisStore[15].Axis[1..15].Pos18.Reached := FALSE;
   AxisStore[1].Axis[1..15].Pos19.Position := 0.0;
   AxisStore[2].Axis[1..15].Pos19.Position := 0.0;
   AxisStore[3].Axis[1..15].Pos19.Position := 0.0;
   AxisStore[4].Axis[1..15].Pos19.Position := 0.0;
   AxisStore[5].Axis[1..15].Pos19.Position := 0.0;
   AxisStore[6].Axis[1..15].Pos19.Position := 0.0;
   AxisStore[7].Axis[1..15].Pos19.Position := 0.0;
   AxisStore[8].Axis[1..15].Pos19.Position := 0.0;
   AxisStore[9].Axis[1..15].Pos19.Position := 0.0;
   AxisStore[10].Axis[1..15].Pos19.Position := 0.0;
   AxisStore[11].Axis[1..15].Pos19.Position := 0.0;
   AxisStore[12].Axis[1..15].Pos19.Position := 0.0;
   AxisStore[13].Axis[1..15].Pos19.Position := 0.0;
   AxisStore[14].Axis[1..15].Pos19.Position := 0.0;
   AxisStore[15].Axis[1..15].Pos19.Position := 0.0;
   AxisStore[1].Axis[1..15].Pos19.Speed := 0;
   AxisStore[2].Axis[1..15].Pos19.Speed := 0;
   AxisStore[3].Axis[1..15].Pos19.Speed := 0;
   AxisStore[4].Axis[1..15].Pos19.Speed := 0;
   AxisStore[5].Axis[1..15].Pos19.Speed := 0;
   AxisStore[6].Axis[1..15].Pos19.Speed := 0;
   AxisStore[7].Axis[1..15].Pos19.Speed := 0;
   AxisStore[8].Axis[1..15].Pos19.Speed := 0;
   AxisStore[9].Axis[1..15].Pos19.Speed := 0;
   AxisStore[10].Axis[1..15].Pos19.Speed := 0;
   AxisStore[11].Axis[1..15].Pos19.Speed := 0;
   AxisStore[12].Axis[1..15].Pos19.Speed := 0;
   AxisStore[13].Axis[1..15].Pos19.Speed := 0;
   AxisStore[14].Axis[1..15].Pos19.Speed := 0;
   AxisStore[15].Axis[1..15].Pos19.Speed := 0;
   AxisStore[1].Axis[1..15].Pos19.Reached := FALSE;
   AxisStore[2].Axis[1..15].Pos19.Reached := FALSE;
   AxisStore[3].Axis[1..15].Pos19.Reached := FALSE;
   AxisStore[4].Axis[1..15].Pos19.Reached := FALSE;
   AxisStore[5].Axis[1..15].Pos19.Reached := FALSE;
   AxisStore[6].Axis[1..15].Pos19.Reached := FALSE;
   AxisStore[7].Axis[1..15].Pos19.Reached := FALSE;
   AxisStore[8].Axis[1..15].Pos19.Reached := FALSE;
   AxisStore[9].Axis[1..15].Pos19.Reached := FALSE;
   AxisStore[10].Axis[1..15].Pos19.Reached := FALSE;
   AxisStore[11].Axis[1..15].Pos19.Reached := FALSE;
   AxisStore[12].Axis[1..15].Pos19.Reached := FALSE;
   AxisStore[13].Axis[1..15].Pos19.Reached := FALSE;
   AxisStore[14].Axis[1..15].Pos19.Reached := FALSE;
   AxisStore[15].Axis[1..15].Pos19.Reached := FALSE;
   AxisStore[1].Axis[1..15].Pos20.Position := 0.0;
   AxisStore[2].Axis[1..15].Pos20.Position := 0.0;
   AxisStore[3].Axis[1..15].Pos20.Position := 0.0;
   AxisStore[4].Axis[1..15].Pos20.Position := 0.0;
   AxisStore[5].Axis[1..15].Pos20.Position := 0.0;
   AxisStore[6].Axis[1..15].Pos20.Position := 0.0;
   AxisStore[7].Axis[1..15].Pos20.Position := 0.0;
   AxisStore[8].Axis[1..15].Pos20.Position := 0.0;
   AxisStore[9].Axis[1..15].Pos20.Position := 0.0;
   AxisStore[10].Axis[1..15].Pos20.Position := 0.0;
   AxisStore[11].Axis[1..15].Pos20.Position := 0.0;
   AxisStore[12].Axis[1..15].Pos20.Position := 0.0;
   AxisStore[13].Axis[1..15].Pos20.Position := 0.0;
   AxisStore[14].Axis[1..15].Pos20.Position := 0.0;
   AxisStore[15].Axis[1..15].Pos20.Position := 0.0;
   AxisStore[1].Axis[1..15].Pos20.Speed := 0;
   AxisStore[2].Axis[1..15].Pos20.Speed := 0;
   AxisStore[3].Axis[1..15].Pos20.Speed := 0;
   AxisStore[4].Axis[1..15].Pos20.Speed := 0;
   AxisStore[5].Axis[1..15].Pos20.Speed := 0;
   AxisStore[6].Axis[1..15].Pos20.Speed := 0;
   AxisStore[7].Axis[1..15].Pos20.Speed := 0;
   AxisStore[8].Axis[1..15].Pos20.Speed := 0;
   AxisStore[9].Axis[1..15].Pos20.Speed := 0;
   AxisStore[10].Axis[1..15].Pos20.Speed := 0;
   AxisStore[11].Axis[1..15].Pos20.Speed := 0;
   AxisStore[12].Axis[1..15].Pos20.Speed := 0;
   AxisStore[13].Axis[1..15].Pos20.Speed := 0;
   AxisStore[14].Axis[1..15].Pos20.Speed := 0;
   AxisStore[15].Axis[1..15].Pos20.Speed := 0;
   AxisStore[1].Axis[1..15].Pos20.Reached := FALSE;
   AxisStore[2].Axis[1..15].Pos20.Reached := FALSE;
   AxisStore[3].Axis[1..15].Pos20.Reached := FALSE;
   AxisStore[4].Axis[1..15].Pos20.Reached := FALSE;
   AxisStore[5].Axis[1..15].Pos20.Reached := FALSE;
   AxisStore[6].Axis[1..15].Pos20.Reached := FALSE;
   AxisStore[7].Axis[1..15].Pos20.Reached := FALSE;
   AxisStore[8].Axis[1..15].Pos20.Reached := FALSE;
   AxisStore[9].Axis[1..15].Pos20.Reached := FALSE;
   AxisStore[10].Axis[1..15].Pos20.Reached := FALSE;
   AxisStore[11].Axis[1..15].Pos20.Reached := FALSE;
   AxisStore[12].Axis[1..15].Pos20.Reached := FALSE;
   AxisStore[13].Axis[1..15].Pos20.Reached := FALSE;
   AxisStore[14].Axis[1..15].Pos20.Reached := FALSE;
   AxisStore[15].Axis[1..15].Pos20.Reached := FALSE;
   AxisStore[1].Axis[1..15].Pos21.Position := 0.0;
   AxisStore[2].Axis[1..15].Pos21.Position := 0.0;
   AxisStore[3].Axis[1..15].Pos21.Position := 0.0;
   AxisStore[4].Axis[1..15].Pos21.Position := 0.0;
   AxisStore[5].Axis[1..15].Pos21.Position := 0.0;
   AxisStore[6].Axis[1..15].Pos21.Position := 0.0;
   AxisStore[7].Axis[1..15].Pos21.Position := 0.0;
   AxisStore[8].Axis[1..15].Pos21.Position := 0.0;
   AxisStore[9].Axis[1..15].Pos21.Position := 0.0;
   AxisStore[10].Axis[1..15].Pos21.Position := 0.0;
   AxisStore[11].Axis[1..15].Pos21.Position := 0.0;
   AxisStore[12].Axis[1..15].Pos21.Position := 0.0;
   AxisStore[13].Axis[1..15].Pos21.Position := 0.0;
   AxisStore[14].Axis[1..15].Pos21.Position := 0.0;
   AxisStore[15].Axis[1..15].Pos21.Position := 0.0;
   AxisStore[1].Axis[1..15].Pos21.Speed := 0;
   AxisStore[2].Axis[1..15].Pos21.Speed := 0;
   AxisStore[3].Axis[1..15].Pos21.Speed := 0;
   AxisStore[4].Axis[1..15].Pos21.Speed := 0;
   AxisStore[5].Axis[1..15].Pos21.Speed := 0;
   AxisStore[6].Axis[1..15].Pos21.Speed := 0;
   AxisStore[7].Axis[1..15].Pos21.Speed := 0;
   AxisStore[8].Axis[1..15].Pos21.Speed := 0;
   AxisStore[9].Axis[1..15].Pos21.Speed := 0;
   AxisStore[10].Axis[1..15].Pos21.Speed := 0;
   AxisStore[11].Axis[1..15].Pos21.Speed := 0;
   AxisStore[12].Axis[1..15].Pos21.Speed := 0;
   AxisStore[13].Axis[1..15].Pos21.Speed := 0;
   AxisStore[14].Axis[1..15].Pos21.Speed := 0;
   AxisStore[15].Axis[1..15].Pos21.Speed := 0;
   AxisStore[1].Axis[1..15].Pos21.Reached := FALSE;
   AxisStore[2].Axis[1..15].Pos21.Reached := FALSE;
   AxisStore[3].Axis[1..15].Pos21.Reached := FALSE;
   AxisStore[4].Axis[1..15].Pos21.Reached := FALSE;
   AxisStore[5].Axis[1..15].Pos21.Reached := FALSE;
   AxisStore[6].Axis[1..15].Pos21.Reached := FALSE;
   AxisStore[7].Axis[1..15].Pos21.Reached := FALSE;
   AxisStore[8].Axis[1..15].Pos21.Reached := FALSE;
   AxisStore[9].Axis[1..15].Pos21.Reached := FALSE;
   AxisStore[10].Axis[1..15].Pos21.Reached := FALSE;
   AxisStore[11].Axis[1..15].Pos21.Reached := FALSE;
   AxisStore[12].Axis[1..15].Pos21.Reached := FALSE;
   AxisStore[13].Axis[1..15].Pos21.Reached := FALSE;
   AxisStore[14].Axis[1..15].Pos21.Reached := FALSE;
   AxisStore[15].Axis[1..15].Pos21.Reached := FALSE;
   AxisStore[1].Axis[1..15].Pos22.Position := 0.0;
   AxisStore[2].Axis[1..15].Pos22.Position := 0.0;
   AxisStore[3].Axis[1..15].Pos22.Position := 0.0;
   AxisStore[4].Axis[1..15].Pos22.Position := 0.0;
   AxisStore[5].Axis[1..15].Pos22.Position := 0.0;
   AxisStore[6].Axis[1..15].Pos22.Position := 0.0;
   AxisStore[7].Axis[1..15].Pos22.Position := 0.0;
   AxisStore[8].Axis[1..15].Pos22.Position := 0.0;
   AxisStore[9].Axis[1..15].Pos22.Position := 0.0;
   AxisStore[10].Axis[1..15].Pos22.Position := 0.0;
   AxisStore[11].Axis[1..15].Pos22.Position := 0.0;
   AxisStore[12].Axis[1..15].Pos22.Position := 0.0;
   AxisStore[13].Axis[1..15].Pos22.Position := 0.0;
   AxisStore[14].Axis[1..15].Pos22.Position := 0.0;
   AxisStore[15].Axis[1..15].Pos22.Position := 0.0;
   AxisStore[1].Axis[1..15].Pos22.Speed := 0;
   AxisStore[2].Axis[1..15].Pos22.Speed := 0;
   AxisStore[3].Axis[1..15].Pos22.Speed := 0;
   AxisStore[4].Axis[1..15].Pos22.Speed := 0;
   AxisStore[5].Axis[1..15].Pos22.Speed := 0;
   AxisStore[6].Axis[1..15].Pos22.Speed := 0;
   AxisStore[7].Axis[1..15].Pos22.Speed := 0;
   AxisStore[8].Axis[1..15].Pos22.Speed := 0;
   AxisStore[9].Axis[1..15].Pos22.Speed := 0;
   AxisStore[10].Axis[1..15].Pos22.Speed := 0;
   AxisStore[11].Axis[1..15].Pos22.Speed := 0;
   AxisStore[12].Axis[1..15].Pos22.Speed := 0;
   AxisStore[13].Axis[1..15].Pos22.Speed := 0;
   AxisStore[14].Axis[1..15].Pos22.Speed := 0;
   AxisStore[15].Axis[1..15].Pos22.Speed := 0;
   AxisStore[1].Axis[1..15].Pos22.Reached := FALSE;
   AxisStore[2].Axis[1..15].Pos22.Reached := FALSE;
   AxisStore[3].Axis[1..15].Pos22.Reached := FALSE;
   AxisStore[4].Axis[1..15].Pos22.Reached := FALSE;
   AxisStore[5].Axis[1..15].Pos22.Reached := FALSE;
   AxisStore[6].Axis[1..15].Pos22.Reached := FALSE;
   AxisStore[7].Axis[1..15].Pos22.Reached := FALSE;
   AxisStore[8].Axis[1..15].Pos22.Reached := FALSE;
   AxisStore[9].Axis[1..15].Pos22.Reached := FALSE;
   AxisStore[10].Axis[1..15].Pos22.Reached := FALSE;
   AxisStore[11].Axis[1..15].Pos22.Reached := FALSE;
   AxisStore[12].Axis[1..15].Pos22.Reached := FALSE;
   AxisStore[13].Axis[1..15].Pos22.Reached := FALSE;
   AxisStore[14].Axis[1..15].Pos22.Reached := FALSE;
   AxisStore[15].Axis[1..15].Pos22.Reached := FALSE;
   AxisStore[1].Axis[1..15].Pos23.Position := 0.0;
   AxisStore[2].Axis[1..15].Pos23.Position := 0.0;
   AxisStore[3].Axis[1..15].Pos23.Position := 0.0;
   AxisStore[4].Axis[1..15].Pos23.Position := 0.0;
   AxisStore[5].Axis[1..15].Pos23.Position := 0.0;
   AxisStore[6].Axis[1..15].Pos23.Position := 0.0;
   AxisStore[7].Axis[1..15].Pos23.Position := 0.0;
   AxisStore[8].Axis[1..15].Pos23.Position := 0.0;
   AxisStore[9].Axis[1..15].Pos23.Position := 0.0;
   AxisStore[10].Axis[1..15].Pos23.Position := 0.0;
   AxisStore[11].Axis[1..15].Pos23.Position := 0.0;
   AxisStore[12].Axis[1..15].Pos23.Position := 0.0;
   AxisStore[13].Axis[1..15].Pos23.Position := 0.0;
   AxisStore[14].Axis[1..15].Pos23.Position := 0.0;
   AxisStore[15].Axis[1..15].Pos23.Position := 0.0;
   AxisStore[1].Axis[1..15].Pos23.Speed := 0;
   AxisStore[2].Axis[1..15].Pos23.Speed := 0;
   AxisStore[3].Axis[1..15].Pos23.Speed := 0;
   AxisStore[4].Axis[1..15].Pos23.Speed := 0;
   AxisStore[5].Axis[1..15].Pos23.Speed := 0;
   AxisStore[6].Axis[1..15].Pos23.Speed := 0;
   AxisStore[7].Axis[1..15].Pos23.Speed := 0;
   AxisStore[8].Axis[1..15].Pos23.Speed := 0;
   AxisStore[9].Axis[1..15].Pos23.Speed := 0;
   AxisStore[10].Axis[1..15].Pos23.Speed := 0;
   AxisStore[11].Axis[1..15].Pos23.Speed := 0;
   AxisStore[12].Axis[1..15].Pos23.Speed := 0;
   AxisStore[13].Axis[1..15].Pos23.Speed := 0;
   AxisStore[14].Axis[1..15].Pos23.Speed := 0;
   AxisStore[15].Axis[1..15].Pos23.Speed := 0;
   AxisStore[1].Axis[1..15].Pos23.Reached := FALSE;
   AxisStore[2].Axis[1..15].Pos23.Reached := FALSE;
   AxisStore[3].Axis[1..15].Pos23.Reached := FALSE;
   AxisStore[4].Axis[1..15].Pos23.Reached := FALSE;
   AxisStore[5].Axis[1..15].Pos23.Reached := FALSE;
   AxisStore[6].Axis[1..15].Pos23.Reached := FALSE;
   AxisStore[7].Axis[1..15].Pos23.Reached := FALSE;
   AxisStore[8].Axis[1..15].Pos23.Reached := FALSE;
   AxisStore[9].Axis[1..15].Pos23.Reached := FALSE;
   AxisStore[10].Axis[1..15].Pos23.Reached := FALSE;
   AxisStore[11].Axis[1..15].Pos23.Reached := FALSE;
   AxisStore[12].Axis[1..15].Pos23.Reached := FALSE;
   AxisStore[13].Axis[1..15].Pos23.Reached := FALSE;
   AxisStore[14].Axis[1..15].Pos23.Reached := FALSE;
   AxisStore[15].Axis[1..15].Pos23.Reached := FALSE;
   AxisStore[1].Axis[1..15].Pos24.Position := 0.0;
   AxisStore[2].Axis[1..15].Pos24.Position := 0.0;
   AxisStore[3].Axis[1..15].Pos24.Position := 0.0;
   AxisStore[4].Axis[1..15].Pos24.Position := 0.0;
   AxisStore[5].Axis[1..15].Pos24.Position := 0.0;
   AxisStore[6].Axis[1..15].Pos24.Position := 0.0;
   AxisStore[7].Axis[1..15].Pos24.Position := 0.0;
   AxisStore[8].Axis[1..15].Pos24.Position := 0.0;
   AxisStore[9].Axis[1..15].Pos24.Position := 0.0;
   AxisStore[10].Axis[1..15].Pos24.Position := 0.0;
   AxisStore[11].Axis[1..15].Pos24.Position := 0.0;
   AxisStore[12].Axis[1..15].Pos24.Position := 0.0;
   AxisStore[13].Axis[1..15].Pos24.Position := 0.0;
   AxisStore[14].Axis[1..15].Pos24.Position := 0.0;
   AxisStore[15].Axis[1..15].Pos24.Position := 0.0;
   AxisStore[1].Axis[1..15].Pos24.Speed := 0;
   AxisStore[2].Axis[1..15].Pos24.Speed := 0;
   AxisStore[3].Axis[1..15].Pos24.Speed := 0;
   AxisStore[4].Axis[1..15].Pos24.Speed := 0;
   AxisStore[5].Axis[1..15].Pos24.Speed := 0;
   AxisStore[6].Axis[1..15].Pos24.Speed := 0;
   AxisStore[7].Axis[1..15].Pos24.Speed := 0;
   AxisStore[8].Axis[1..15].Pos24.Speed := 0;
   AxisStore[9].Axis[1..15].Pos24.Speed := 0;
   AxisStore[10].Axis[1..15].Pos24.Speed := 0;
   AxisStore[11].Axis[1..15].Pos24.Speed := 0;
   AxisStore[12].Axis[1..15].Pos24.Speed := 0;
   AxisStore[13].Axis[1..15].Pos24.Speed := 0;
   AxisStore[14].Axis[1..15].Pos24.Speed := 0;
   AxisStore[15].Axis[1..15].Pos24.Speed := 0;
   AxisStore[1].Axis[1..15].Pos24.Reached := FALSE;
   AxisStore[2].Axis[1..15].Pos24.Reached := FALSE;
   AxisStore[3].Axis[1..15].Pos24.Reached := FALSE;
   AxisStore[4].Axis[1..15].Pos24.Reached := FALSE;
   AxisStore[5].Axis[1..15].Pos24.Reached := FALSE;
   AxisStore[6].Axis[1..15].Pos24.Reached := FALSE;
   AxisStore[7].Axis[1..15].Pos24.Reached := FALSE;
   AxisStore[8].Axis[1..15].Pos24.Reached := FALSE;
   AxisStore[9].Axis[1..15].Pos24.Reached := FALSE;
   AxisStore[10].Axis[1..15].Pos24.Reached := FALSE;
   AxisStore[11].Axis[1..15].Pos24.Reached := FALSE;
   AxisStore[12].Axis[1..15].Pos24.Reached := FALSE;
   AxisStore[13].Axis[1..15].Pos24.Reached := FALSE;
   AxisStore[14].Axis[1..15].Pos24.Reached := FALSE;
   AxisStore[15].Axis[1..15].Pos24.Reached := FALSE;
   AxisStore[1].Axis[1..15].Pos25.Position := 0.0;
   AxisStore[2].Axis[1..15].Pos25.Position := 0.0;
   AxisStore[3].Axis[1..15].Pos25.Position := 0.0;
   AxisStore[4].Axis[1..15].Pos25.Position := 0.0;
   AxisStore[5].Axis[1..15].Pos25.Position := 0.0;
   AxisStore[6].Axis[1..15].Pos25.Position := 0.0;
   AxisStore[7].Axis[1..15].Pos25.Position := 0.0;
   AxisStore[8].Axis[1..15].Pos25.Position := 0.0;
   AxisStore[9].Axis[1..15].Pos25.Position := 0.0;
   AxisStore[10].Axis[1..15].Pos25.Position := 0.0;
   AxisStore[11].Axis[1..15].Pos25.Position := 0.0;
   AxisStore[12].Axis[1..15].Pos25.Position := 0.0;
   AxisStore[13].Axis[1..15].Pos25.Position := 0.0;
   AxisStore[14].Axis[1..15].Pos25.Position := 0.0;
   AxisStore[15].Axis[1..15].Pos25.Position := 0.0;
   AxisStore[1].Axis[1..15].Pos25.Speed := 0;
   AxisStore[2].Axis[1..15].Pos25.Speed := 0;
   AxisStore[3].Axis[1..15].Pos25.Speed := 0;
   AxisStore[4].Axis[1..15].Pos25.Speed := 0;
   AxisStore[5].Axis[1..15].Pos25.Speed := 0;
   AxisStore[6].Axis[1..15].Pos25.Speed := 0;
   AxisStore[7].Axis[1..15].Pos25.Speed := 0;
   AxisStore[8].Axis[1..15].Pos25.Speed := 0;
   AxisStore[9].Axis[1..15].Pos25.Speed := 0;
   AxisStore[10].Axis[1..15].Pos25.Speed := 0;
   AxisStore[11].Axis[1..15].Pos25.Speed := 0;
   AxisStore[12].Axis[1..15].Pos25.Speed := 0;
   AxisStore[13].Axis[1..15].Pos25.Speed := 0;
   AxisStore[14].Axis[1..15].Pos25.Speed := 0;
   AxisStore[15].Axis[1..15].Pos25.Speed := 0;
   AxisStore[1].Axis[1..15].Pos25.Reached := FALSE;
   AxisStore[2].Axis[1..15].Pos25.Reached := FALSE;
   AxisStore[3].Axis[1..15].Pos25.Reached := FALSE;
   AxisStore[4].Axis[1..15].Pos25.Reached := FALSE;
   AxisStore[5].Axis[1..15].Pos25.Reached := FALSE;
   AxisStore[6].Axis[1..15].Pos25.Reached := FALSE;
   AxisStore[7].Axis[1..15].Pos25.Reached := FALSE;
   AxisStore[8].Axis[1..15].Pos25.Reached := FALSE;
   AxisStore[9].Axis[1..15].Pos25.Reached := FALSE;
   AxisStore[10].Axis[1..15].Pos25.Reached := FALSE;
   AxisStore[11].Axis[1..15].Pos25.Reached := FALSE;
   AxisStore[12].Axis[1..15].Pos25.Reached := FALSE;
   AxisStore[13].Axis[1..15].Pos25.Reached := FALSE;
   AxisStore[14].Axis[1..15].Pos25.Reached := FALSE;
   AxisStore[15].Axis[1..15].Pos25.Reached := FALSE;
   AxisStore[1].Axis[1..15].Pos26.Position := 0.0;
   AxisStore[2].Axis[1..15].Pos26.Position := 0.0;
   AxisStore[3].Axis[1..15].Pos26.Position := 0.0;
   AxisStore[4].Axis[1..15].Pos26.Position := 0.0;
   AxisStore[5].Axis[1..15].Pos26.Position := 0.0;
   AxisStore[6].Axis[1..15].Pos26.Position := 0.0;
   AxisStore[7].Axis[1..15].Pos26.Position := 0.0;
   AxisStore[8].Axis[1..15].Pos26.Position := 0.0;
   AxisStore[9].Axis[1..15].Pos26.Position := 0.0;
   AxisStore[10].Axis[1..15].Pos26.Position := 0.0;
   AxisStore[11].Axis[1..15].Pos26.Position := 0.0;
   AxisStore[12].Axis[1..15].Pos26.Position := 0.0;
   AxisStore[13].Axis[1..15].Pos26.Position := 0.0;
   AxisStore[14].Axis[1..15].Pos26.Position := 0.0;
   AxisStore[15].Axis[1..15].Pos26.Position := 0.0;
   AxisStore[1].Axis[1..15].Pos26.Speed := 0;
   AxisStore[2].Axis[1..15].Pos26.Speed := 0;
   AxisStore[3].Axis[1..15].Pos26.Speed := 0;
   AxisStore[4].Axis[1..15].Pos26.Speed := 0;
   AxisStore[5].Axis[1..15].Pos26.Speed := 0;
   AxisStore[6].Axis[1..15].Pos26.Speed := 0;
   AxisStore[7].Axis[1..15].Pos26.Speed := 0;
   AxisStore[8].Axis[1..15].Pos26.Speed := 0;
   AxisStore[9].Axis[1..15].Pos26.Speed := 0;
   AxisStore[10].Axis[1..15].Pos26.Speed := 0;
   AxisStore[11].Axis[1..15].Pos26.Speed := 0;
   AxisStore[12].Axis[1..15].Pos26.Speed := 0;
   AxisStore[13].Axis[1..15].Pos26.Speed := 0;
   AxisStore[14].Axis[1..15].Pos26.Speed := 0;
   AxisStore[15].Axis[1..15].Pos26.Speed := 0;
   AxisStore[1].Axis[1..15].Pos26.Reached := FALSE;
   AxisStore[2].Axis[1..15].Pos26.Reached := FALSE;
   AxisStore[3].Axis[1..15].Pos26.Reached := FALSE;
   AxisStore[4].Axis[1..15].Pos26.Reached := FALSE;
   AxisStore[5].Axis[1..15].Pos26.Reached := FALSE;
   AxisStore[6].Axis[1..15].Pos26.Reached := FALSE;
   AxisStore[7].Axis[1..15].Pos26.Reached := FALSE;
   AxisStore[8].Axis[1..15].Pos26.Reached := FALSE;
   AxisStore[9].Axis[1..15].Pos26.Reached := FALSE;
   AxisStore[10].Axis[1..15].Pos26.Reached := FALSE;
   AxisStore[11].Axis[1..15].Pos26.Reached := FALSE;
   AxisStore[12].Axis[1..15].Pos26.Reached := FALSE;
   AxisStore[13].Axis[1..15].Pos26.Reached := FALSE;
   AxisStore[14].Axis[1..15].Pos26.Reached := FALSE;
   AxisStore[15].Axis[1..15].Pos26.Reached := FALSE;
   AxisStore[1].Axis[1..15].Pos27.Position := 0.0;
   AxisStore[2].Axis[1..15].Pos27.Position := 0.0;
   AxisStore[3].Axis[1..15].Pos27.Position := 0.0;
   AxisStore[4].Axis[1..15].Pos27.Position := 0.0;
   AxisStore[5].Axis[1..15].Pos27.Position := 0.0;
   AxisStore[6].Axis[1..15].Pos27.Position := 0.0;
   AxisStore[7].Axis[1..15].Pos27.Position := 0.0;
   AxisStore[8].Axis[1..15].Pos27.Position := 0.0;
   AxisStore[9].Axis[1..15].Pos27.Position := 0.0;
   AxisStore[10].Axis[1..15].Pos27.Position := 0.0;
   AxisStore[11].Axis[1..15].Pos27.Position := 0.0;
   AxisStore[12].Axis[1..15].Pos27.Position := 0.0;
   AxisStore[13].Axis[1..15].Pos27.Position := 0.0;
   AxisStore[14].Axis[1..15].Pos27.Position := 0.0;
   AxisStore[15].Axis[1..15].Pos27.Position := 0.0;
   AxisStore[1].Axis[1..15].Pos27.Speed := 0;
   AxisStore[2].Axis[1..15].Pos27.Speed := 0;
   AxisStore[3].Axis[1..15].Pos27.Speed := 0;
   AxisStore[4].Axis[1..15].Pos27.Speed := 0;
   AxisStore[5].Axis[1..15].Pos27.Speed := 0;
   AxisStore[6].Axis[1..15].Pos27.Speed := 0;
   AxisStore[7].Axis[1..15].Pos27.Speed := 0;
   AxisStore[8].Axis[1..15].Pos27.Speed := 0;
   AxisStore[9].Axis[1..15].Pos27.Speed := 0;
   AxisStore[10].Axis[1..15].Pos27.Speed := 0;
   AxisStore[11].Axis[1..15].Pos27.Speed := 0;
   AxisStore[12].Axis[1..15].Pos27.Speed := 0;
   AxisStore[13].Axis[1..15].Pos27.Speed := 0;
   AxisStore[14].Axis[1..15].Pos27.Speed := 0;
   AxisStore[15].Axis[1..15].Pos27.Speed := 0;
   AxisStore[1].Axis[1..15].Pos27.Reached := FALSE;
   AxisStore[2].Axis[1..15].Pos27.Reached := FALSE;
   AxisStore[3].Axis[1..15].Pos27.Reached := FALSE;
   AxisStore[4].Axis[1..15].Pos27.Reached := FALSE;
   AxisStore[5].Axis[1..15].Pos27.Reached := FALSE;
   AxisStore[6].Axis[1..15].Pos27.Reached := FALSE;
   AxisStore[7].Axis[1..15].Pos27.Reached := FALSE;
   AxisStore[8].Axis[1..15].Pos27.Reached := FALSE;
   AxisStore[9].Axis[1..15].Pos27.Reached := FALSE;
   AxisStore[10].Axis[1..15].Pos27.Reached := FALSE;
   AxisStore[11].Axis[1..15].Pos27.Reached := FALSE;
   AxisStore[12].Axis[1..15].Pos27.Reached := FALSE;
   AxisStore[13].Axis[1..15].Pos27.Reached := FALSE;
   AxisStore[14].Axis[1..15].Pos27.Reached := FALSE;
   AxisStore[15].Axis[1..15].Pos27.Reached := FALSE;
   AxisStore[1].Axis[1..15].Pos28.Position := 0.0;
   AxisStore[2].Axis[1..15].Pos28.Position := 0.0;
   AxisStore[3].Axis[1..15].Pos28.Position := 0.0;
   AxisStore[4].Axis[1..15].Pos28.Position := 0.0;
   AxisStore[5].Axis[1..15].Pos28.Position := 0.0;
   AxisStore[6].Axis[1..15].Pos28.Position := 0.0;
   AxisStore[7].Axis[1..15].Pos28.Position := 0.0;
   AxisStore[8].Axis[1..15].Pos28.Position := 0.0;
   AxisStore[9].Axis[1..15].Pos28.Position := 0.0;
   AxisStore[10].Axis[1..15].Pos28.Position := 0.0;
   AxisStore[11].Axis[1..15].Pos28.Position := 0.0;
   AxisStore[12].Axis[1..15].Pos28.Position := 0.0;
   AxisStore[13].Axis[1..15].Pos28.Position := 0.0;
   AxisStore[14].Axis[1..15].Pos28.Position := 0.0;
   AxisStore[15].Axis[1..15].Pos28.Position := 0.0;
   AxisStore[1].Axis[1..15].Pos28.Speed := 0;
   AxisStore[2].Axis[1..15].Pos28.Speed := 0;
   AxisStore[3].Axis[1..15].Pos28.Speed := 0;
   AxisStore[4].Axis[1..15].Pos28.Speed := 0;
   AxisStore[5].Axis[1..15].Pos28.Speed := 0;
   AxisStore[6].Axis[1..15].Pos28.Speed := 0;
   AxisStore[7].Axis[1..15].Pos28.Speed := 0;
   AxisStore[8].Axis[1..15].Pos28.Speed := 0;
   AxisStore[9].Axis[1..15].Pos28.Speed := 0;
   AxisStore[10].Axis[1..15].Pos28.Speed := 0;
   AxisStore[11].Axis[1..15].Pos28.Speed := 0;
   AxisStore[12].Axis[1..15].Pos28.Speed := 0;
   AxisStore[13].Axis[1..15].Pos28.Speed := 0;
   AxisStore[14].Axis[1..15].Pos28.Speed := 0;
   AxisStore[15].Axis[1..15].Pos28.Speed := 0;
   AxisStore[1].Axis[1..15].Pos28.Reached := FALSE;
   AxisStore[2].Axis[1..15].Pos28.Reached := FALSE;
   AxisStore[3].Axis[1..15].Pos28.Reached := FALSE;
   AxisStore[4].Axis[1..15].Pos28.Reached := FALSE;
   AxisStore[5].Axis[1..15].Pos28.Reached := FALSE;
   AxisStore[6].Axis[1..15].Pos28.Reached := FALSE;
   AxisStore[7].Axis[1..15].Pos28.Reached := FALSE;
   AxisStore[8].Axis[1..15].Pos28.Reached := FALSE;
   AxisStore[9].Axis[1..15].Pos28.Reached := FALSE;
   AxisStore[10].Axis[1..15].Pos28.Reached := FALSE;
   AxisStore[11].Axis[1..15].Pos28.Reached := FALSE;
   AxisStore[12].Axis[1..15].Pos28.Reached := FALSE;
   AxisStore[13].Axis[1..15].Pos28.Reached := FALSE;
   AxisStore[14].Axis[1..15].Pos28.Reached := FALSE;
   AxisStore[15].Axis[1..15].Pos28.Reached := FALSE;
   AxisStore[1].Axis[1..15].Pos29.Position := 0.0;
   AxisStore[2].Axis[1..15].Pos29.Position := 0.0;
   AxisStore[3].Axis[1..15].Pos29.Position := 0.0;
   AxisStore[4].Axis[1..15].Pos29.Position := 0.0;
   AxisStore[5].Axis[1..15].Pos29.Position := 0.0;
   AxisStore[6].Axis[1..15].Pos29.Position := 0.0;
   AxisStore[7].Axis[1..15].Pos29.Position := 0.0;
   AxisStore[8].Axis[1..15].Pos29.Position := 0.0;
   AxisStore[9].Axis[1..15].Pos29.Position := 0.0;
   AxisStore[10].Axis[1..15].Pos29.Position := 0.0;
   AxisStore[11].Axis[1..15].Pos29.Position := 0.0;
   AxisStore[12].Axis[1..15].Pos29.Position := 0.0;
   AxisStore[13].Axis[1..15].Pos29.Position := 0.0;
   AxisStore[14].Axis[1..15].Pos29.Position := 0.0;
   AxisStore[15].Axis[1..15].Pos29.Position := 0.0;
   AxisStore[1].Axis[1..15].Pos29.Speed := 0;
   AxisStore[2].Axis[1..15].Pos29.Speed := 0;
   AxisStore[3].Axis[1..15].Pos29.Speed := 0;
   AxisStore[4].Axis[1..15].Pos29.Speed := 0;
   AxisStore[5].Axis[1..15].Pos29.Speed := 0;
   AxisStore[6].Axis[1..15].Pos29.Speed := 0;
   AxisStore[7].Axis[1..15].Pos29.Speed := 0;
   AxisStore[8].Axis[1..15].Pos29.Speed := 0;
   AxisStore[9].Axis[1..15].Pos29.Speed := 0;
   AxisStore[10].Axis[1..15].Pos29.Speed := 0;
   AxisStore[11].Axis[1..15].Pos29.Speed := 0;
   AxisStore[12].Axis[1..15].Pos29.Speed := 0;
   AxisStore[13].Axis[1..15].Pos29.Speed := 0;
   AxisStore[14].Axis[1..15].Pos29.Speed := 0;
   AxisStore[15].Axis[1..15].Pos29.Speed := 0;
   AxisStore[1].Axis[1..15].Pos29.Reached := FALSE;
   AxisStore[2].Axis[1..15].Pos29.Reached := FALSE;
   AxisStore[3].Axis[1..15].Pos29.Reached := FALSE;
   AxisStore[4].Axis[1..15].Pos29.Reached := FALSE;
   AxisStore[5].Axis[1..15].Pos29.Reached := FALSE;
   AxisStore[6].Axis[1..15].Pos29.Reached := FALSE;
   AxisStore[7].Axis[1..15].Pos29.Reached := FALSE;
   AxisStore[8].Axis[1..15].Pos29.Reached := FALSE;
   AxisStore[9].Axis[1..15].Pos29.Reached := FALSE;
   AxisStore[10].Axis[1..15].Pos29.Reached := FALSE;
   AxisStore[11].Axis[1..15].Pos29.Reached := FALSE;
   AxisStore[12].Axis[1..15].Pos29.Reached := FALSE;
   AxisStore[13].Axis[1..15].Pos29.Reached := FALSE;
   AxisStore[14].Axis[1..15].Pos29.Reached := FALSE;
   AxisStore[15].Axis[1..15].Pos29.Reached := FALSE;
   AxisStore[1].Axis[1..15].Pos30.Position := 0.0;
   AxisStore[2].Axis[1..15].Pos30.Position := 0.0;
   AxisStore[3].Axis[1..15].Pos30.Position := 0.0;
   AxisStore[4].Axis[1..15].Pos30.Position := 0.0;
   AxisStore[5].Axis[1..15].Pos30.Position := 0.0;
   AxisStore[6].Axis[1..15].Pos30.Position := 0.0;
   AxisStore[7].Axis[1..15].Pos30.Position := 0.0;
   AxisStore[8].Axis[1..15].Pos30.Position := 0.0;
   AxisStore[9].Axis[1..15].Pos30.Position := 0.0;
   AxisStore[10].Axis[1..15].Pos30.Position := 0.0;
   AxisStore[11].Axis[1..15].Pos30.Position := 0.0;
   AxisStore[12].Axis[1..15].Pos30.Position := 0.0;
   AxisStore[13].Axis[1..15].Pos30.Position := 0.0;
   AxisStore[14].Axis[1..15].Pos30.Position := 0.0;
   AxisStore[15].Axis[1..15].Pos30.Position := 0.0;
   AxisStore[1].Axis[1..15].Pos30.Speed := 0;
   AxisStore[2].Axis[1..15].Pos30.Speed := 0;
   AxisStore[3].Axis[1..15].Pos30.Speed := 0;
   AxisStore[4].Axis[1..15].Pos30.Speed := 0;
   AxisStore[5].Axis[1..15].Pos30.Speed := 0;
   AxisStore[6].Axis[1..15].Pos30.Speed := 0;
   AxisStore[7].Axis[1..15].Pos30.Speed := 0;
   AxisStore[8].Axis[1..15].Pos30.Speed := 0;
   AxisStore[9].Axis[1..15].Pos30.Speed := 0;
   AxisStore[10].Axis[1..15].Pos30.Speed := 0;
   AxisStore[11].Axis[1..15].Pos30.Speed := 0;
   AxisStore[12].Axis[1..15].Pos30.Speed := 0;
   AxisStore[13].Axis[1..15].Pos30.Speed := 0;
   AxisStore[14].Axis[1..15].Pos30.Speed := 0;
   AxisStore[15].Axis[1..15].Pos30.Speed := 0;
   AxisStore[1].Axis[1..15].Pos30.Reached := FALSE;
   AxisStore[2].Axis[1..15].Pos30.Reached := FALSE;
   AxisStore[3].Axis[1..15].Pos30.Reached := FALSE;
   AxisStore[4].Axis[1..15].Pos30.Reached := FALSE;
   AxisStore[5].Axis[1..15].Pos30.Reached := FALSE;
   AxisStore[6].Axis[1..15].Pos30.Reached := FALSE;
   AxisStore[7].Axis[1..15].Pos30.Reached := FALSE;
   AxisStore[8].Axis[1..15].Pos30.Reached := FALSE;
   AxisStore[9].Axis[1..15].Pos30.Reached := FALSE;
   AxisStore[10].Axis[1..15].Pos30.Reached := FALSE;
   AxisStore[11].Axis[1..15].Pos30.Reached := FALSE;
   AxisStore[12].Axis[1..15].Pos30.Reached := FALSE;
   AxisStore[13].Axis[1..15].Pos30.Reached := FALSE;
   AxisStore[14].Axis[1..15].Pos30.Reached := FALSE;
   AxisStore[15].Axis[1..15].Pos30.Reached := FALSE;
END_DATA_BLOCK
